ABB RAPID module: FSNA0464C.mod

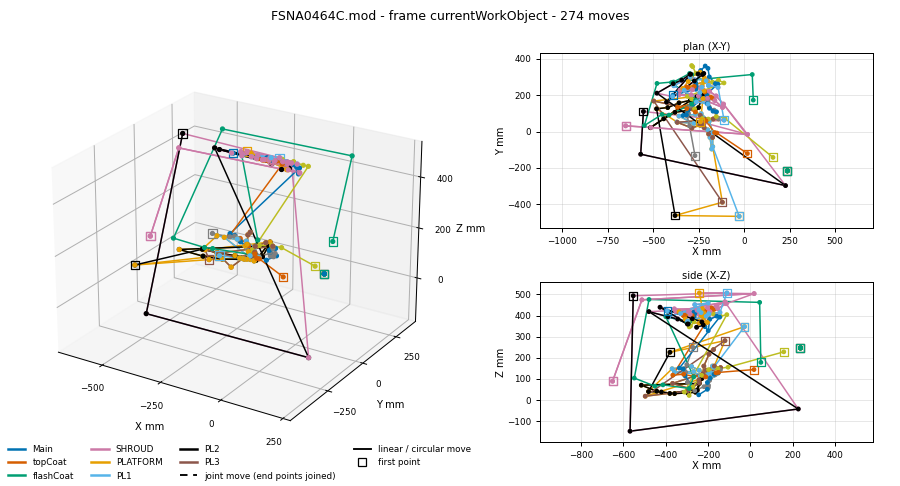
[picture p0: tool path of FSNA0464C.mod in frame currentWorkObject, 274 of 274 moves have a stored position in this frame; points joined in program order, loops and branches not executed]
MODULE FSNA0464C

    ! 10-10-24
    !
    ! declare and/or define variables that are local to this module
    LOCAL CONST listitem partProgram{3}:=[["","TopCoat"],["","FlashCoat"],[stEmpty,"Stop"]];
    LOCAL VAR string defaultValueString;
    VAR num itemselected:=0;
    VAR buttondata buttonAnswer:=0;
    LOCAL VAR robtarget pInt_temp1;
	PERS zonedata pathairfoil:=[FALSE,100,100,100,75,75,15];
    !
    VAR num myTemp := 0;
    VAR num X_Shift := 0;
    VAR num X_Value := 0;
    VAR num Y_Shift := 0;
    VAR num Y_Value := 0;
    VAR num Z_Shift := 0;
    VAR num Z_Value := 0;
    VAR num Speed := 0;
    VAR num LargestDistance := 0;
    VAR num numberOfLines := 0;
    VAR num FirstPass := 0;
    !
    ! positions for Airfoil CTARR
    CONST robtarget p1:=[[-480.99,124.94,40.31],[0.241886,0.571759,0.755176,0.210457],[0,1,1,0],[0,67.5741,9E+9,9E+9,9E+9,9E+9]];
    CONST robtarget p2:=[[-419.82,131.58,38.25],[0.241885,0.571758,0.755177,0.210457],[0,1,1,0],[0,59.8741,9E+9,9E+9,9E+9,9E+9]];
    CONST robtarget p3:=[[-357.80,157.50,30.89],[0.25135,0.552212,0.746055,0.274387],[0,1,1,0],[0,49.8741,9E+9,9E+9,9E+9,9E+9]];
    CONST robtarget p4:=[[-295.67,171.59,34.02],[0.258412,0.447595,0.729271,0.448381],[0,1,1,0],[0,44.2741,9E+9,9E+9,9E+9,9E+9]];
    CONST robtarget p5:=[[-258.93,192.30,37.24],[0.258413,0.447594,0.729271,0.448381],[0,1,1,0],[0,30.6741,9E+9,9E+9,9E+9,9E+9]];
    CONST robtarget p6:=[[-240.79,207.18,79.11],[0.336518,0.448757,0.687079,0.461839],[0,1,1,0],[0,18.4741,9E+9,9E+9,9E+9,9E+9]];
    CONST robtarget p7:=[[1532.27,28.26,128.24],[0.245924,0.528851,0.800385,-0.138642],[0,0,0,0],[0,558.621,9E+9,9E+9,9E+9,9E+9]];
    CONST robtarget p8:=[[-514.99,21.05,70.50],[0.286821,0.504649,0.813028,0.0452658],[0,1,1,0],[0,67.5741,9E+9,9E+9,9E+9,9E+9]];
    CONST robtarget p9:=[[-441.94,69.98,41.95],[0.327155,0.53741,0.777145,0.0143071],[0,1,1,0],[0,59.8741,9E+9,9E+9,9E+9,9E+9]];
    CONST robtarget p10:=[[-380.23,105.47,31.38],[0.392331,0.6189,0.675982,0.078028],[0,2,1,0],[0,49.8741,9E+9,9E+9,9E+9,9E+9]];
    !
    CONST robtarget p11:=[[-268.27,122.31,50.17],[0.448624,0.648801,0.591368,0.167566],[0,2,1,0],[0,44.2741,9E+9,9E+9,9E+9,9E+9]];
    CONST robtarget p12:=[[-250.17,131.85,47.00],[0.481979,0.715929,0.422761,0.276432],[0,2,1,0],[0,30.6741,9E+9,9E+9,9E+9,9E+9]];
    CONST robtarget p13:=[[-229.13,197.03,101.76],[0.452914,0.539488,0.537819,0.463219],[0,1,1,0],[0,24.4741,9E+9,9E+9,9E+9,9E+9]];
    CONST robtarget p14:=[[1816.81,23.63,146.28],[0.530012,0.0601364,0.839977,0.0995457],[-1,0,-1,0],[0,485.704,9E+9,9E+9,9E+9,9E+9]];
    CONST robtarget p15:=[[1496.69,-77.72,540],[0.712477,-0.0505666,0.699591,0.0197792],[-1,-1,-1,0],[120.002,9E+09,9E+09,9E+09,9E+09,9E+09]];
    CONST robtarget p16:=[[1503.37,67.93,540],[0.712477,-0.0505667,0.699591,0.0197793],[-1,-1,-1,0],[150.003,9E+09,9E+09,9E+09,9E+09,9E+09]];
    CONST robtarget p17:=[[1525.14,108.88,540],[0.712477,-0.0505668,0.699591,0.0197793],[-1,-1,-1,0],[195.004,9E+09,9E+09,9E+09,9E+09,9E+09]];
    CONST robtarget p18:=[[1539.77,199.84,540],[0.712477,-0.0505668,0.699591,0.0197793],[-1,-1,-1,0],[230.001,9E+09,9E+09,9E+09,9E+09,9E+09]];
    CONST robtarget p19:=[[-172.56,-82.90,154.81],[0.0598896,-0.960037,0.272975,-0.0150686],[0,-1,2,0],[0,162.3,9E+9,9E+9,9E+9,9E+9]];
    CONST robtarget p20:=[[-172.53,-7.13,117.30],[0.0598902,-0.960037,0.272975,-0.0150687],[0,-1,2,0],[0,164,9E+9,9E+9,9E+9,9E+9]];
    !
    CONST robtarget p21:=[[-191.10,57.42,100.93],[0.0655881,-0.94736,0.311192,-0.0369689],[0,-1,2,0],[0,173.5,9E+9,9E+9,9E+9,9E+9]];
    CONST robtarget p22:=[[-236.16,98.35,113.48],[0.0598898,-0.960037,0.272975,-0.0150686],[0,-1,2,0],[0,188.8,9E+9,9E+9,9E+9,9E+9]];
    CONST robtarget p23:=[[-267.77,93.84,135.02],[0.0372043,-0.989337,0.123334,0.0679511],[0,-1,2,0],[0,200.8,9E+9,9E+9,9E+9,9E+9]];
    CONST robtarget p24:=[[-358.18,84.85,132.45],[0.0372035,-0.989337,0.123334,0.0679511],[0,-1,2,0],[0,209.5,9E+9,9E+9,9E+9,9E+9]];
    CONST robtarget p25:=[[-172.53,-7.13,117.30],[0.0598902,-0.960037,0.272975,-0.0150687],[0,-1,2,0],[0,164,9E+9,9E+9,9E+9,9E+9]];
    CONST robtarget p26:=[[-178.25,-95.93,161.15],[0.0598899,-0.960037,0.272975,-0.0150685],[0,-1,2,0],[0,162.3,9E+9,9E+9,9E+9,9E+9]];
    CONST robtarget p27:=[[-187.56,-32.42,129.52],[0.0598899,-0.960037,0.272975,-0.0150687],[0,-1,2,0],[0,164,9E+9,9E+9,9E+9,9E+9]];
    CONST robtarget p28:=[[-200.37,9.66,124.39],[0.065588,-0.94736,0.311192,-0.0369689],[0,-1,2,0],[0,173.5,9E+9,9E+9,9E+9,9E+9]];
    CONST robtarget p29:=[[-241.64,42.37,141.08],[0.05989,-0.960037,0.272975,-0.0150686],[0,-1,2,0],[0,188.8,9E+9,9E+9,9E+9,9E+9]];
    CONST robtarget p30:=[[-277.12,44.60,159.21],[0.037204,-0.989337,0.123334,0.0679512],[0,-1,2,0],[0,200.8,9E+9,9E+9,9E+9,9E+9]];
    !
    CONST robtarget p31:=[[-369.35,52.61,148.19],[0.0372036,-0.989337,0.123334,0.0679511],[0,-1,2,0],[0,209.5,9E+9,9E+9,9E+9,9E+9]];
    CONST robtarget p32:=[[1621.31,158.58,690],[0.712477,-0.0505667,0.699591,0.0197792],[-1,-1,-1,0],[-0.00322896,9E+09,9E+09,9E+09,9E+09,9E+09]];
    CONST robtarget p33:=[[1620.84,58.68,700],[0.712477,-0.0505667,0.699591,0.0197793],[-1,-1,-1,0],[9.9958,9E+09,9E+09,9E+09,9E+09,9E+09]];
    CONST robtarget p34:=[[1665.7,-160.7,700],[0.712477,-0.0505667,0.699591,0.0197793],[-1,-1,-1,0],[70.0029,9E+09,9E+09,9E+09,9E+09,9E+09]];
    CONST robtarget p35:=[[1496.69,-77.72,700],[0.712477,-0.0505666,0.699591,0.0197792],[-1,-1,-1,0],[120.002,9E+09,9E+09,9E+09,9E+09,9E+09]];
    CONST robtarget p36:=[[1503.37,67.93,690],[0.712477,-0.0505667,0.699591,0.0197793],[-1,-1,-1,0],[150.003,9E+09,9E+09,9E+09,9E+09,9E+09]];
    CONST robtarget p37:=[[1525.14,108.88,690],[0.712477,-0.0505668,0.699591,0.0197793],[-1,-1,-1,0],[195.004,9E+09,9E+09,9E+09,9E+09,9E+09]];
    CONST robtarget p38:=[[1539.77,199.84,700],[0.712477,-0.0505668,0.699591,0.0197793],[-1,-1,-1,0],[230.001,9E+09,9E+09,9E+09,9E+09,9E+09]];
    CONST robtarget p39:=[[1444.86,284.59,700],[0.712477,-0.0505668,0.699591,0.0197793],[0,-1,-1,0],[270.004,9E+09,9E+09,9E+09,9E+09,9E+09]];
    CONST robtarget p40:=[[-496.31,167.54,18.41],[0.302398,0.557141,0.772704,0.0328229],[0,1,1,0],[0,35.3741,9E+9,9E+9,9E+9,9E+9]];
    !
    CONST robtarget p41:=[[-296.07,126.18,42.89],[0.3024,0.55714,0.772704,0.0328239],[0,1,1,0],[0,25.4741,9E+9,9E+9,9E+9,9E+9]];
    CONST robtarget p42:=[[-240.83,89.12,81.91],[0.302399,0.557141,0.772704,0.0328236],[-1,1,1,0],[0,4.4741,9E+9,9E+9,9E+9,9E+9]];
    CONST robtarget p43:=[[-215.91,67.47,112.59],[0.302399,0.557141,0.772704,0.0328236],[-1,1,1,0],[0,-9.7259,9E+9,9E+9,9E+9,9E+9]];
    CONST robtarget p44:=[[-208.79,59.37,141.39],[0.302399,0.557141,0.772704,0.0328237],[-1,1,1,0],[0,-25.4259,9E+9,9E+9,9E+9,9E+9]];
    CONST robtarget p45:=[[-169.72,69.14,160.90],[0.302399,0.557141,0.772704,0.0328238],[-1,1,1,0],[0,-33.5259,9E+9,9E+9,9E+9,9E+9]];
    CONST robtarget p46:=[[-140.26,69.36,153.83],[0.302399,0.55714,0.772704,0.0328239],[-1,1,1,0],[0,-42.5259,9E+9,9E+9,9E+9,9E+9]];
    CONST robtarget p48:=[[-366.97,50.44,78.97],[0.302398,0.557141,0.772704,0.0328232],[0,1,1,0],[0,35.3741,9E+9,9E+9,9E+9,9E+9]];
    CONST robtarget p49:=[[-287.06,19.27,54.47],[0.302399,0.557141,0.772704,0.032823],[-1,1,1,0],[0,25.4741,9E+9,9E+9,9E+9,9E+9]];

    PERS robtarget p201:=[[-190.59,221.15,418.28],[0.323876,-0.134268,0.48472,0.801326],[-1,1,0,0],[0,-184.719,9E+9,9E+9,9E+9,9E+9]];
    PERS robtarget p202:=[[-238.99,240.86,403.58],[0.323876,-0.134268,0.48472,0.801326],[-1,1,0,0],[0,-184.719,9E+9,9E+9,9E+9,9E+9]];
    PERS robtarget p203:=[[-283.49,230.19,405.56],[0.323876,-0.134268,0.48472,0.801326],[-1,1,0,0],[0,-184.719,9E+9,9E+9,9E+9,9E+9]];
    PERS robtarget p204:=[[-351.84,227.15,419.55],[0.323876,-0.134268,0.48472,0.801326],[-1,1,0,0],[0,-184.719,9E+9,9E+9,9E+9,9E+9]];
    PERS robtarget p205:=[[-138.38,318.26,282.97],[0.820959,-0.00154933,0.553533,0.14009],[0,2,-2,0],[0,-333.4,9E+9,9E+9,9E+9,9E+9]];
    PERS robtarget p206:=[[1522.85,30.49,127.90],[0.693528,-0.018539,0.719901,0.0204515],[-1,-1,-1,0],[0,525.079,9E+9,9E+9,9E+9,9E+9]];
    PERS robtarget p207:=[[1533.71,58.37,146.07],[0.688077,-0.0919601,0.714028,0.0908723],[-1,-1,-1,0],[0,525.079,9E+9,9E+9,9E+9,9E+9]];
    PERS robtarget p208:=[[-118.63,132.39,464.09],[0.341814,-0.118033,0.331132,0.871541],[-1,1,0,0],[0,-184.719,9E+9,9E+9,9E+9,9E+9]];
    PERS robtarget p209:=[[-161.24,170.27,444.44],[0.34262,-0.116882,0.321021,0.875155],[-1,1,0,0],[0,-184.719,9E+9,9E+9,9E+9,9E+9]];
    PERS robtarget p210:=[[-201.32,182.62,436.33],[0.342259,-0.117406,0.32561,0.873529],[-1,1,0,0],[0,-184.719,9E+9,9E+9,9E+9,9E+9]];
    !
    PERS robtarget p211:=[[-251.52,195.90,424.71],[0.34323,-0.11596,0.312977,0.877948],[-1,1,0,0],[0,-184.719,9E+9,9E+9,9E+9,9E+9]];
    PERS robtarget p212:=[[-291.38,201.77,418.66],[0.342305,-0.117339,0.325025,0.873738],[-1,1,0,0],[0,-184.719,9E+9,9E+9,9E+9,9E+9]];
    PERS robtarget p213:=[[-358.88,201.75,431.17],[0.34234,-0.11729,0.324591,0.873892],[-1,1,0,0],[0,-184.719,9E+9,9E+9,9E+9,9E+9]];
    PERS robtarget p214:=[[1526.81,49.01,147.72],[0.53358,0.309144,0.772491,-0.151589],[0,0,0,0],[0,525.079,9E+9,9E+9,9E+9,9E+9]];
    PERS robtarget p215:=[[-141.45,-101.58,920.03],[0.650986,0.194184,0.706774,-0.197436],[-1,0,0,0],[82.817,9E+09,9E+09,9E+09,9E+09,9E+09]];
    PERS robtarget p216:=[[-88.05,-18.09,920.70],[0.650993,0.194178,0.706763,-0.197458],[0,0,0,0],[82.817,9E+09,9E+09,9E+09,9E+09,9E+09]];
    PERS robtarget p217:=[[-21.87,98.95,918.25],[0.65099,0.194168,0.706777,-0.197427],[0,0,0,0],[82.817,9E+09,9E+09,9E+09,9E+09,9E+09]];
    PERS robtarget p218:=[[53.24,222.48,897.26],[0.65098,0.194179,0.706786,-0.197419],[0,0,0,0],[82.817,9E+09,9E+09,9E+09,9E+09,9E+09]];
    PERS robtarget p219:=[[45.58,94.46,899.85],[0.0855565,0.697288,0.707868,-0.0734352],[0,0,0,0],[104.005,9E+09,9E+09,9E+09,9E+09,9E+09]];
    PERS robtarget p220:=[[-221.03,177.90,433.71],[0.343488,0.0801029,0.438498,0.826631],[-1,1,0,0],[0,-140.019,9E+9,9E+9,9E+9,9E+9]];
    !
    PERS robtarget p221:=[[-226.19,180.94,432.49],[0.55509,0.111637,0.37794,0.732512],[0,1,0,0],[0,-140.019,9E+9,9E+9,9E+9,9E+9]];
    PERS robtarget p222:=[[-219.63,223.62,412.03],[0.561411,0.0905932,0.427662,0.702649],[0,1,0,0],[0,-140.019,9E+9,9E+9,9E+9,9E+9]];
    PERS robtarget p223:=[[-230.74,249.72,398.97],[0.562161,0.0874597,0.434857,0.698015],[0,1,0,0],[0,-140.019,9E+9,9E+9,9E+9,9E+9]];
    PERS robtarget p224:=[[-220.10,274.50,389.30],[0.52604,0.192483,0.577288,0.594113],[0,1,0,0],[0,-140.019,9E+9,9E+9,9E+9,9E+9]];
    PERS robtarget p225:=[[-202.24,278.15,367.26],[0.464891,0.348117,0.609092,0.540091],[0,1,1,0],[0,-140.019,9E+9,9E+9,9E+9,9E+9]];
    PERS robtarget p226:=[[1608.55,16.90,696.10],[0.496587,-0.139785,0.281765,-0.808993],[0,-1,1,0],[25.0035,9E+9,9E+9,9E+9,9E+9,9E+9]];
    PERS robtarget p227:=[[1502.42,-81.35,694.68],[0.496587,-0.139785,0.281765,-0.808993],[0,-1,1,0],[0,9E+9,9E+9,9E+9,9E+9,9E+9]];
    PERS robtarget p228:=[[1461.90,-160.07,687.75],[0.496587,-0.139785,0.281765,-0.808993],[0,-1,1,0],[-0.000826709,9E+9,9E+9,9E+9,9E+9,9E+9]];
    !
    PERS robtarget p231:=[[-293.61,298.88,371.24],[0.0151509,-0.0827354,0.608731,0.788906],[-1,0,0,0],[0,-140.019,9E+9,9E+9,9E+9,9E+9]];
    PERS robtarget p232:=[[-241.43,325.70,363.53],[0.174125,0.0732031,0.694697,0.694059],[-1,0,0,0],[0,-140.019,9E+9,9E+9,9E+9,9E+9]];
    PERS robtarget p233:=[[-219.10,295.28,358.44],[0.464891,0.348117,0.609092,0.540091],[0,1,1,0],[0,-140.019,9E+9,9E+9,9E+9,9E+9]];
    PERS robtarget p234:=[[1381.21,176.71,690.45],[0.509919,-0.0782388,0.181097,-0.837296],[0,-1,1,0],[74.9967,9E+9,9E+9,9E+9,9E+9,9E+9]];
    PERS robtarget p235:=[[1460.37,118.23,690.06],[0.505886,-0.101083,0.218555,-0.828308],[0,-1,1,0],[49.9958,9E+9,9E+9,9E+9,9E+9,9E+9]];
    PERS robtarget p236:=[[1453.88,16.90,696.10],[0.496587,-0.139785,0.281765,-0.808993],[0,-1,1,0],[25.0035,9E+9,9E+9,9E+9,9E+9,9E+9]];
    PERS robtarget p237:=[[1308.94,-160.07,687.75],[0.496587,-0.139785,0.281765,-0.808993],[0,-1,1,0],[-0.000826709,9E+9,9E+9,9E+9,9E+9,9E+9]];
    PERS robtarget p238:=[[1411.45,-160.07,687.75],[0.496587,-0.139785,0.281765,-0.808993],[0,-1,1,0],[-0.000826709,9E+9,9E+9,9E+9,9E+9,9E+9]];
    !
    PERS robtarget p241:=[[1858.30,301.74,499.76],[0.179089,0.917392,0.34153,0.0983641],[0,1,0,0],[-175.061,9E+9,9E+9,9E+9,9E+9,9E+9]];
    PERS robtarget p242:=[[1614.86,199.00,509.29],[0.175594,0.951771,0.23609,0.086952],[0,1,-1,0],[-190.061,9E+9,9E+9,9E+9,9E+9,9E+9]];
    PERS robtarget p243:=[[1502.55,134.04,503.05],[0.185136,0.908581,0.362955,0.0920279],[0,1,0,0],[-220.061,9E+9,9E+9,9E+9,9E+9,9E+9]];
    PERS robtarget p244:=[[1494.58,104.81,490.86],[0.174159,0.800358,0.560783,0.120907],[0,1,0,0],[-240.061,9E+9,9E+9,9E+9,9E+9,9E+9]];
    PERS robtarget p245:=[[1559.49,159.93,488.36],[0.149738,0.674434,0.699604,0.182406],[0,1,0,0],[-310.061,9E+9,9E+9,9E+9,9E+9,9E+9]];
    PERS robtarget p246:=[[1600.54,33.00,493.44],[0.172748,0.593565,0.769913,0.158344],[-1,0,0,0],[-330.061,9E+9,9E+9,9E+9,9E+9,9E+9]];
    PERS robtarget p247:=[[1500.24,-78.88,512.52],[0.130233,0.625317,0.75886,0.12708],[-1,0,0,0],[-350.061,9E+9,9E+9,9E+9,9E+9,9E+9]];
    PERS robtarget p248:=[[1338.41,-93.31,512.24],[0.126705,0.803062,0.571687,0.110503],[-1,1,0,0],[-375.061,9E+9,9E+9,9E+9,9E+9,9E+9]];
    !

    ! declare and/or define position variables that are local to this module
	PERS robtarget home:=[[114.84,-94.02,-57.43],[0.398229,-0.576485,0.66735,0.252432],[-1,-1,-1,0],[0,372.2,9E+9,9E+9,9E+9,9E+9]];
	PERS robtarget pounce:=[[114.84,-94.02,-57.43],[0.398229,-0.576485,0.66735,0.252432],[-1,-1,-1,0],[0,0,9E+9,9E+9,9E+9,9E+9]];
    PERS robtarget home10:=[[-37.25,141.01,1171.15],[0.656992,0.226174,0.64921,-0.309408],[0,-1,0,0],[-0.00177226,9E+09,9E+09,9E+09,9E+09,9E+09]];
    PERS robtarget home20:=[[-47.87,162.56,920.76],[0.566373,0.264704,0.729584,-0.277237],[0,0,0,0],[0.0306373,9E+09,9E+09,9E+09,9E+09,9E+09]];
    PERS robtarget pounce10:=[[1506.92,-117.30,148.10],[0.362896,-0.228602,0.902396,0.0415831],[-1,-1,-1,0],[0,-6.2069,9E+9,9E+9,9E+9,9E+9]];
    PERS robtarget mypounce:=[[-379.47,-461.24,226.09],[0.186927,-0.20553,0.960411,0.0206579],[-1,0,1,0],[0,162.3,9E+9,9E+9,9E+9,9E+9]];
    PERS robtarget mypounce10:=[[-27.24,-465.79,347.27],[0.059889,-0.960037,0.272975,-0.0150683],[-1,-1,2,0],[0,162.3,9E+9,9E+9,9E+9,9E+9]];
    PERS robtarget mypounce20:=[[-119.56,-388.27,281.05],[0.286821,0.504649,0.813028,0.0452658],[-1,1,1,0],[0,67.5741,9E+9,9E+9,9E+9,9E+9]];
    PERS robtarget mypounce30:=[[158.59,-142.09,228.20],[0.41173,-0.607554,0.614434,0.289531],[-1,-1,1,0],[0,-21.0832,9E+9,9E+9,9E+9,9E+9]];
    PERS robtarget mypounce40:=[[-391.18,199.72,419.59],[0.346718,-0.644484,0.557145,0.39245],[0,-1,1,0],[0,-99.7753,9E+9,9E+9,9E+9,9E+9]];
    PERS robtarget mypounce50:=[[17.77,-120.71,144.39],[0.403174,-0.614096,0.639379,0.227004],[-1,-1,2,0],[0,-195,9E+9,9E+9,9E+9,9E+9]];
    PERS wobjdata wobj1:=[FALSE,TRUE,"",[[0,0,0],[1,0,0,0]],[[1526.4,-255.043,47.4813],[0.766931,0.185105,-0.133095,-0.599865]]];
    PERS robtarget p0:=[[1402.40,207.74,74.69],[0.420282,-0.489062,0.761608,-0.0643041],[0,-1,0,0],[0,453.104,9E+9,9E+9,9E+9,9E+9]];
    PERS robtarget mypounce60:=[[50.15,172.68,178.39],[0.441257,-0.541665,0.672728,0.243575],[-1,0,1,0],[0,-286.004,9E+9,9E+9,9E+9,9E+9]];
    PERS robtarget tempval:=[[1776.74,50.33,181.37],[0.419919,-0.484892,0.74874,-0.167142],[-1,-1,0,0],[0,453.104,9E+9,9E+9,9E+9,9E+9]];
    PERS robtarget tempval10:=[[1776.74,50.33,181.37],[0.419919,-0.484892,0.74874,-0.167142],[-1,-1,0,0],[0,453.104,9E+9,9E+9,9E+9,9E+9]];
    PERS robtarget mypouncePL:=[[1450.05,-296.49,158.45],[0.000887637,0.674822,0.737972,0.00347664],[-1,0,0,0],[0,368.4,9E+9,9E+9,9E+9,9E+9]];
    PERS robtarget mypouncePL10:=[[1453.74,-212.15,169.09],[0.000887898,0.674822,0.737972,0.00347632],[-1,0,0,0],[0,368.4,9E+9,9E+9,9E+9,9E+9]];
    PERS robtarget p50:=[[-242.82,35.16,96.19],[0.302399,0.557141,0.772704,0.0328234],[-1,1,1,0],[0,4.4741,9E+9,9E+9,9E+9,9E+9]];
    PERS robtarget p60:=[[-104.77,71.85,155.57],[0.235728,-0.65255,0.702889,0.15671],[-1,-1,1,0],[0,-21.0832,9E+9,9E+9,9E+9,9E+9]];
    PERS robtarget p70:=[[-223.35,269.54,407.36],[0.490279,-0.512469,0.629658,0.317069],[0,0,2,0],[0,-21.0832,9E+9,9E+9,9E+9,9E+9]];
    PERS robtarget p51:=[[-224.08,37.20,124.71],[0.302399,0.557141,0.772704,0.0328239],[-1,1,1,0],[0,-9.7259,9E+9,9E+9,9E+9,9E+9]];
    PERS robtarget p53:=[[-195.00,-13.72,216.84],[0.302399,0.55714,0.772704,0.0328239],[-1,1,1,0],[0,-33.5259,9E+9,9E+9,9E+9,9E+9]];
    PERS robtarget p52:=[[-219.36,20.60,161.04],[0.302399,0.557141,0.772704,0.0328233],[-1,1,1,0],[0,-25.4259,9E+9,9E+9,9E+9,9E+9]];
    PERS robtarget p54:=[[-173.44,-32.53,238.99],[0.302399,0.55714,0.772704,0.0328235],[-1,1,1,0],[0,-42.5259,9E+9,9E+9,9E+9,9E+9]];
    PERS robtarget p55:=[[1627.55,-144.85,103.80],[0.37608,-0.272238,0.874139,0.142592],[-1,-1,-1,0],[0,473.679,9E+9,9E+9,9E+9,9E+9]];
    PERS robtarget p56:=[[1636.24,-58.87,104.20],[0.37057,-0.304807,0.863301,0.156466],[-1,-1,-1,0],[0,473.679,9E+9,9E+9,9E+9,9E+9]];
    PERS robtarget p57:=[[1542.81,-38.49,90.01],[0.365729,-0.330862,0.853641,0.167539],[-1,-1,-1,0],[0,473.679,9E+9,9E+9,9E+9,9E+9]];
    PERS robtarget p58:=[[1415.80,3.28,64.46],[0.365729,-0.330862,0.853641,0.167539],[-1,-1,-1,0],[0,473.679,9E+9,9E+9,9E+9,9E+9]];
    PERS robtarget p67:=[[-110.76,267.07,404.11],[0.363074,-0.624312,0.643864,0.252685],[-1,-1,1,0],[0,-21.0832,9E+9,9E+9,9E+9,9E+9]];
    PERS robtarget p61:=[[-152.80,82.65,148.87],[0.187257,-0.658057,0.719316,0.120335],[0,-1,1,0],[0,-21.0832,9E+9,9E+9,9E+9,9E+9]];
    PERS robtarget p62:=[[-197.09,68.49,143.85],[0.187257,-0.658057,0.719316,0.120335],[0,-1,1,0],[0,-21.0832,9E+9,9E+9,9E+9,9E+9]];
    PERS robtarget p63:=[[-229.45,71.30,117.03],[0.227436,-0.599619,0.763307,0.0780525],[0,0,2,0],[0,-21.0832,9E+9,9E+9,9E+9,9E+9]];
    PERS robtarget p80:=[[-265.55,232.07,416.89],[0.144535,-0.701198,0.368316,0.593105],[-1,0,1,0],[0,-99.7753,9E+9,9E+9,9E+9,9E+9]];
    PERS robtarget p81:=[[-261.58,246.21,409.97],[0.144535,-0.701198,0.368316,0.593105],[-1,0,1,0],[0,-99.7753,9E+9,9E+9,9E+9,9E+9]];
    PERS robtarget p82:=[[-265.06,264.67,396.52],[0.144535,-0.701198,0.368316,0.593105],[-1,0,1,0],[0,-99.7753,9E+9,9E+9,9E+9,9E+9]];
    PERS robtarget p83:=[[-238.77,335.25,363.62],[0.339406,-0.656714,0.470947,0.481392],[-1,-1,1,0],[0,-99.7753,9E+9,9E+9,9E+9,9E+9]];
    PERS robtarget p93:=[[-202.77,199.89,50.99],[0.336532,-0.904926,0.260301,-0.00990511],[0,-1,2,0],[0,-99.7753,9E+9,9E+9,9E+9,9E+9]];
    PERS robtarget p103:=[[-267.84,107.34,111.99],[0.393028,-0.576819,0.672319,0.246569],[0,0,2,0],[0,-195,9E+9,9E+9,9E+9,9E+9]];
    PERS robtarget p94:=[[-202.59,152.76,83.34],[0.304048,-0.849853,0.395123,-0.170828],[0,-1,2,0],[0,-99.7753,9E+9,9E+9,9E+9,9E+9]];
    PERS robtarget p84:=[[-213.83,359.92,347.10],[0.394944,-0.635518,0.506567,0.4284],[-1,-1,1,0],[0,-99.7753,9E+9,9E+9,9E+9,9E+9]];
    PERS robtarget p85:=[[-198.67,346.90,328.05],[0.475693,-0.58931,0.583419,0.293345],[0,-1,2,0],[0,-99.7753,9E+9,9E+9,9E+9,9E+9]];
    PERS robtarget p95:=[[-190.25,127.73,103.49],[0.304048,-0.849853,0.395123,-0.170828],[0,-1,2,0],[0,-99.7753,9E+9,9E+9,9E+9,9E+9]];
    PERS robtarget p105:=[[-366.09,132.79,118.09],[0.323041,-0.635333,0.624263,0.319831],[0,-1,1,0],[0,-195,9E+9,9E+9,9E+9,9E+9]];
    PERS robtarget p86:=[[-191.26,300.09,382.38],[0.59614,-0.483857,0.607528,0.203491],[0,-1,2,0],[0,-99.7753,9E+9,9E+9,9E+9,9E+9]];
    PERS robtarget p87:=[[-157.75,263.05,396.69],[0.59614,-0.483857,0.607528,0.203491],[0,-1,2,0],[0,-99.7753,9E+9,9E+9,9E+9,9E+9]];
    PERS robtarget p97:=[[-151.71,108.34,127.85],[0.455068,-0.790762,0.388826,-0.128156],[0,-1,2,0],[0,-99.7753,9E+9,9E+9,9E+9,9E+9]];
    PERS robtarget p107:=[[-171.00,182.73,428.83],[0.510833,-0.489852,0.656726,0.260396],[0,0,2,0],[0,-195,9E+9,9E+9,9E+9,9E+9]];
    PERS robtarget p88:=[[-144.63,260.94,392.22],[0.53853,-0.525652,0.641502,0.148831],[0,-1,2,0],[0,-99.7753,9E+9,9E+9,9E+9,9E+9]];
    PERS robtarget p89:=[[-335.05,88.30,151.37],[0.225425,-0.851908,0.331482,0.336981],[0,-1,2,0],[0,-99.7753,9E+9,9E+9,9E+9,9E+9]];
    PERS robtarget p68:=[[-140.93,282.02,396.74],[0.416985,-0.58835,0.652857,0.231831],[0,-1,2,0],[0,-21.0832,9E+9,9E+9,9E+9,9E+9]];
    PERS robtarget p59:=[[1256.15,38.08,77.18],[0.365729,-0.330862,0.853641,0.167539],[-1,-1,-1,0],[0,473.679,9E+9,9E+9,9E+9,9E+9]];
    PERS robtarget p47:=[[1532.27,28.26,128.24],[0.245924,0.528851,0.800385,-0.138642],[0,0,0,0],[0,558.621,9E+9,9E+9,9E+9,9E+9]];
    PERS robtarget p90:=[[-316.97,91.92,146.99],[0.220546,-0.85345,0.324574,0.342979],[-1,-1,2,0],[0,-99.7753,9E+9,9E+9,9E+9,9E+9]];
    PERS robtarget p66:=[[-311.42,193.18,37.97],[0.305868,-0.633875,0.658667,0.266093],[0,-1,1,0],[0,-21.0832,9E+9,9E+9,9E+9,9E+9]];
    PERS robtarget p64:=[[-272.18,123.81,60.95],[0.271775,-0.59184,0.749775,0.117051],[0,0,2,0],[0,-21.0832,9E+9,9E+9,9E+9,9E+9]];
    PERS robtarget p65:=[[-288.87,179.42,22.10],[0.318069,-0.603467,0.699672,0.212409],[0,0,2,0],[0,-21.0832,9E+9,9E+9,9E+9,9E+9]];
    PERS robtarget p69:=[[-175.57,271.09,407.55],[0.490279,-0.512469,0.629658,0.317069],[0,0,2,0],[0,-21.0832,9E+9,9E+9,9E+9,9E+9]];
    PERS robtarget p71:=[[-265.49,320.04,370.00],[0.469908,-0.52339,0.645441,0.29775],[0,0,2,0],[0,-21.0832,9E+9,9E+9,9E+9,9E+9]];
    PERS robtarget p72:=[[-282.33,355.82,350.44],[0.500121,-0.506862,0.621602,0.326466],[0,0,2,0],[0,-21.0832,9E+9,9E+9,9E+9,9E+9]];
    PERS robtarget p73:=[[-288.32,362.58,346.09],[0.324166,-0.650206,0.573552,0.3784],[0,-1,1,0],[0,-21.0832,9E+9,9E+9,9E+9,9E+9]];
    PERS robtarget home30:=[[237.33,-215.55,246.81],[0.488992,-0.630948,0.551207,0.242821],[-1,-1,2,0],[0,0.0198783,9E+9,9E+9,9E+9,9E+9]];
    PERS robtarget mypounce70:=[[-512.28,22.13,474.14],[0.177753,-0.1662,0.259277,0.934643],[-1,1,0,0],[0,-286.004,9E+9,9E+9,9E+9,9E+9]];
    PERS robtarget p92:=[[-243.60,195.18,25.06],[0.170318,-0.924324,0.32307,0.110644],[0,-1,2,0],[0,-99.7753,9E+9,9E+9,9E+9,9E+9]];
    PERS robtarget p102:=[[-210.14,59.62,109.88],[0.401472,-0.568723,0.677656,0.236976],[0,0,2,0],[0,-195,9E+9,9E+9,9E+9,9E+9]];
    PERS robtarget p91:=[[-308.15,116.66,114.63],[0.186778,-0.861437,0.276725,0.382705],[-1,-1,2,0],[0,-99.7753,9E+9,9E+9,9E+9,9E+9]];
    PERS robtarget p100:=[[-150.03,-8.14,130.97],[0.440559,-0.527824,0.70084,0.190087],[0,0,2,0],[0,-195,9E+9,9E+9,9E+9,9E+9]];
    PERS robtarget p101:=[[-162.38,-5.44,129.39],[0.440559,-0.527824,0.70084,0.190087],[0,0,2,0],[0,-195,9E+9,9E+9,9E+9,9E+9]];
    PERS robtarget p104:=[[-314.86,126.21,122.37],[0.323041,-0.635333,0.624263,0.319831],[0,-1,1,0],[0,-195,9E+9,9E+9,9E+9,9E+9]];
    PERS robtarget p106:=[[-129.79,110.40,70.28],[0.403174,-0.614096,0.639379,0.227004],[-1,-1,0,0],[0,-66.5,9E+9,9E+9,9E+9,9E+9]];
    PERS robtarget p108:=[[-183.32,189.82,436.24],[0.510833,-0.489852,0.656726,0.260396],[0,0,2,0],[0,-195,9E+9,9E+9,9E+9,9E+9]];
    PERS robtarget p109:=[[-215.24,218.27,420.10],[0.461021,-0.542852,0.639298,0.289947],[0,0,2,0],[0,-195,9E+9,9E+9,9E+9,9E+9]];
    PERS robtarget p110:=[[-274.07,247.53,399.54],[0.4533,-0.55171,0.633072,0.298923],[0,-1,2,0],[0,-195,9E+9,9E+9,9E+9,9E+9]];
    PERS robtarget p111:=[[-308.35,242.58,400.78],[0.403101,-0.611548,0.566935,0.376966],[0,-1,1,0],[0,-195,9E+9,9E+9,9E+9,9E+9]];
    PERS robtarget p112:=[[-316.07,243.83,398.93],[0.372437,-0.628259,0.548013,0.407754],[0,-1,1,0],[0,-195,9E+9,9E+9,9E+9,9E+9]];
    PERS robtarget p113:=[[-22.45,-122.19,118.26],[0.403174,-0.614096,0.639379,0.227004],[-1,-1,0,0],[0,-195,9E+9,9E+9,9E+9,9E+9]];
    PERS robtarget p123:=[[-266.87,171.99,110.22],[0.39541,-0.58203,0.646346,0.295174],[0,0,2,0],[0,-286.004,9E+9,9E+9,9E+9,9E+9]];
    PERS robtarget p120:=[[-451.03,94.08,66.05],[0.230357,-0.682791,0.531307,0.445472],[0,-1,1,0],[0,-286.004,9E+9,9E+9,9E+9,9E+9]];
    PERS robtarget p121:=[[-412.72,90.37,72.14],[0.202711,-0.694159,0.509558,0.466264],[0,-1,1,0],[0,-286.004,9E+9,9E+9,9E+9,9E+9]];
    PERS robtarget p131:=[[-407.31,65.48,14.57],[0.422742,-0.506784,0.679012,0.321562],[-1,1,-2,0],[0,-282,9E+9,9E+9,9E+9,9E+9]];
    PERS robtarget p122:=[[-288.57,151.17,55.23],[0.31947,-0.636015,0.596851,0.370394],[0,-1,1,0],[0,-286.004,9E+9,9E+9,9E+9,9E+9]];
    PERS robtarget mypounce80:=[[-292.56,139.70,-25.36],[0.403174,-0.614096,0.639379,0.227004],[-1,-1,0,0],[0,-24,9E+9,9E+9,9E+9,9E+9]];
    PERS robtarget tp10:=[[-292.56,139.70,-25.36],[0.403174,-0.614096,0.639379,0.227004],[-1,-1,0,0],[0,-24,9E+9,9E+9,9E+9,9E+9]];
    !
    PERS robtarget mypounce110:=[[-482.41,64.04,89.43],[0.313843,-0.686244,0.567806,0.32889],[-1,-1,-1,0],[0,-31.4,9E+9,9E+9,9E+9,9E+9]];
    PERS robtarget p560:=[[-186.00,20.77,115.70],[0.313843,-0.686244,0.567806,0.32889],[-1,-1,-1,0],[0,-31.4,9E+9,9E+9,9E+9,9E+9]];
    PERS robtarget p561:=[[-186.00,20.77,115.70],[0.313843,-0.686244,0.567806,0.32889],[-1,-1,-1,0],[0,-24.7,9E+9,9E+9,9E+9,9E+9]];
    PERS robtarget p562:=[[-184.82,16.87,78.50],[0.313843,-0.686244,0.567806,0.32889],[-1,-1,-1,0],[0,6,9E+9,9E+9,9E+9,9E+9]];
    PERS robtarget p563:=[[-180.94,54.11,26.07],[0.313843,-0.686244,0.567806,0.32889],[-1,-1,-1,0],[0,60,9E+9,9E+9,9E+9,9E+9]];
    PERS robtarget p564:=[[-216.60,41.81,21.25],[0.313843,-0.686244,0.567806,0.32889],[-1,-1,-1,0],[0,108,9E+9,9E+9,9E+9,9E+9]];
    PERS robtarget p565:=[[-127.38,57.13,98.81],[0.403174,-0.614096,0.639379,0.227004],[-1,-1,0,0],[0,-24.7,9E+9,9E+9,9E+9,9E+9]];
    PERS robtarget p566:=[[-189.86,194.53,362.31],[0.403174,-0.614096,0.639379,0.227004],[-1,-1,-1,0],[0,-24.7,9E+9,9E+9,9E+9,9E+9]];
    PERS robtarget p569:=[[-194.35,212.02,353.83],[0.313843,-0.686244,0.567806,0.32889],[-1,-1,-1,0],[0,6,9E+9,9E+9,9E+9,9E+9]];
    PERS robtarget p567:=[[-175.65,149.52,386.03],[0.313843,-0.686244,0.567806,0.32889],[-1,-1,-1,0],[0,-31.4,9E+9,9E+9,9E+9,9E+9]];
    PERS robtarget p568:=[[-205.18,198.55,359.09],[0.313843,-0.686244,0.567806,0.32889],[-1,-1,-1,0],[0,-24.7,9E+9,9E+9,9E+9,9E+9]];
    PERS robtarget p570:=[[-192.85,243.24,335.35],[0.313843,-0.686244,0.567806,0.32889],[-1,-1,-1,0],[0,60,9E+9,9E+9,9E+9,9E+9]];
    PERS robtarget p571:=[[-228.38,214.17,338.21],[0.344401,-0.678774,0.547989,0.346931],[-1,-1,-1,0],[0,108,9E+9,9E+9,9E+9,9E+9]];
    PERS robtarget mypounce120:=[[-477.64,-74.92,-193.25],[0.313843,-0.686244,0.567806,0.32889],[-1,-1,0,0],[0,-31.4,9E+9,9E+9,9E+9,9E+9]];
    PERS robtarget mypounce130:=[[-59.04,-166.15,-141.34],[0.313843,-0.686244,0.567806,0.32889],[-1,-1,0,0],[0,-31.4,9E+9,9E+9,9E+9,9E+9]];
    PERS robtarget mypounce140:=[[-63.83,-26.70,142.30],[0.313843,-0.686244,0.567806,0.32889],[-1,-1,-1,0],[0,-31.4,9E+9,9E+9,9E+9,9E+9]];
    PERS robtarget mypounce90:=[[-284.25,-46.11,66.24],[0.0193857,-0.784247,0.616476,0.0673647],[-1,-1,-1,0],[0,102,9E+9,9E+9,9E+9,9E+9]];
    PERS robtarget p580:=[[-284.25,-46.11,66.24],[0.0193857,-0.784247,0.616476,0.0673647],[-1,-1,-1,0],[0,102,9E+9,9E+9,9E+9,9E+9]];
    PERS robtarget p589:=[[-284.25,-46.11,66.24],[0.0193857,-0.784247,0.616476,0.0673647],[-1,-1,-1,0],[0,102,9E+9,9E+9,9E+9,9E+9]];
    PERS robtarget p581:=[[-284.25,-46.11,66.24],[0.0193857,-0.784247,0.616476,0.0673647],[-1,-1,-1,0],[0,102,9E+9,9E+9,9E+9,9E+9]];
    PERS robtarget p582:=[[-284.25,-46.11,66.24],[0.0193857,-0.784247,0.616476,0.0673647],[-1,-1,-1,0],[0,102,9E+9,9E+9,9E+9,9E+9]];
    PERS robtarget p583:=[[-284.25,-46.11,66.24],[0.0193857,-0.784247,0.616476,0.0673647],[-1,-1,-1,0],[0,102,9E+9,9E+9,9E+9,9E+9]];
    PERS robtarget p584:=[[-284.25,-46.11,66.24],[0.0193857,-0.784247,0.616476,0.0673647],[-1,-1,-1,0],[0,102,9E+9,9E+9,9E+9,9E+9]];
    PERS robtarget p585:=[[-284.25,-46.11,66.24],[0.0193857,-0.784247,0.616476,0.0673647],[-1,-1,-1,0],[0,102,9E+9,9E+9,9E+9,9E+9]];
    PERS robtarget p586:=[[-284.25,-46.11,66.24],[0.0193857,-0.784247,0.616476,0.0673647],[-1,-1,-1,0],[0,102,9E+9,9E+9,9E+9,9E+9]];
    PERS robtarget p587:=[[-284.25,-46.11,66.24],[0.0193857,-0.784247,0.616476,0.0673647],[-1,-1,-1,0],[0,102,9E+9,9E+9,9E+9,9E+9]];
    PERS robtarget p588:=[[-284.25,-46.11,66.24],[0.0193857,-0.784247,0.616476,0.0673647],[-1,-1,-1,0],[0,102,9E+9,9E+9,9E+9,9E+9]];
    PERS robtarget p590:=[[-284.25,-46.11,66.24],[0.0193857,-0.784247,0.616476,0.0673647],[-1,-1,-1,0],[0,102,9E+9,9E+9,9E+9,9E+9]];
    PERS robtarget p591:=[[-284.25,-46.11,66.24],[0.0193857,-0.784247,0.616476,0.0673647],[-1,-1,-1,0],[0,102,9E+9,9E+9,9E+9,9E+9]];
    PERS robtarget p592:=[[-284.25,-46.11,66.24],[0.0193857,-0.784247,0.616476,0.0673647],[-1,-1,-1,0],[0,102,9E+9,9E+9,9E+9,9E+9]];
    PERS robtarget p593:=[[-284.25,-46.11,66.24],[0.0193857,-0.784247,0.616476,0.0673647],[-1,-1,-1,0],[0,102,9E+9,9E+9,9E+9,9E+9]];
    PERS robtarget mypounce100:=[[18.29,-15.44,503.48],[0.169906,-0.161483,0.329654,0.91454],[-1,0,0,0],[0,-184.719,9E+9,9E+9,9E+9,9E+9]];
    PERS robtarget mypounce150:=[[-650.91,31.30,89.26],[0.116327,-0.124282,0.654165,0.736947],[0,1,0,0],[0,-286.004,9E+9,9E+9,9E+9,9E+9]];
    PERS robtarget p126:=[[-399.05,268.85,394.43],[0.259602,-0.689216,0.461688,0.494401],[-1,-1,1,0],[0,-286.004,9E+9,9E+9,9E+9,9E+9]];
    PERS robtarget p127:=[[-387.38,271.93,393.14],[0.259601,-0.689216,0.461688,0.494401],[-1,-1,1,0],[0,-286.004,9E+9,9E+9,9E+9,9E+9]];
    PERS robtarget p128:=[[-299.50,319.00,366.64],[0.326769,-0.626608,0.575511,0.411549],[0,0,1,0],[0,-286.004,9E+9,9E+9,9E+9,9E+9]];
    PERS robtarget p129:=[[-287.20,311.79,370.99],[0.401395,-0.580915,0.618707,0.344415],[0,0,1,0],[0,-286.004,9E+9,9E+9,9E+9,9E+9]];
    PERS robtarget p251:=[[-131.76,239.79,323.25],[0.659486,-0.28722,0.405018,0.564396],[-1,1,-2,0],[0,-306.3,9E+9,9E+9,9E+9,9E+9]];
    PERS robtarget p261:=[[-131.76,239.79,323.25],[0.659486,-0.28722,0.405018,0.564396],[-1,1,-2,0],[0,-306.3,9E+9,9E+9,9E+9,9E+9]];
    PERS robtarget p200:=[[-154.29,195.35,432.99],[0.323876,-0.134268,0.48472,0.801326],[-1,1,0,0],[0,-184.719,9E+9,9E+9,9E+9,9E+9]];
    PERS robtarget p199:=[[-113.53,150.88,455.82],[0.323876,-0.134268,0.48472,0.801326],[-1,1,0,0],[0,-184.719,9E+9,9E+9,9E+9,9E+9]];
    PERS robtarget mypounce160:=[[-240.26,53.18,506.43],[0.349729,-0.0488935,0.333102,0.874267],[-1,1,0,0],[0,-140.019,9E+9,9E+9,9E+9,9E+9]];
    PERS robtarget p229:=[[-336.78,237.08,417.69],[0.0341496,-0.120948,0.464874,0.876412],[-1,0,0,0],[0,-140.019,9E+9,9E+9,9E+9,9E+9]];
    PERS robtarget p230:=[[-307.13,274.36,383.34],[0.0253369,-0.10342,0.534336,0.838539],[-1,0,0,0],[0,-140.019,9E+9,9E+9,9E+9,9E+9]];
    PERS robtarget mypounce170:=[[-110.25,62.51,506.70],[0.0786297,-0.0971196,0.466016,0.875907],[-1,0,0,0],[0,-56.6292,9E+9,9E+9,9E+9,9E+9]];

    PERS robtarget p262:=[[-479.13,210.77,418.40],[0.376944,-0.165729,0.405226,0.816235],[0,1,0,0],[0,72.809,9E+9,9E+9,9E+9,9E+9]];
    PERS robtarget p263:=[[-389.18,262.86,394.40],[0.376944,-0.165729,0.405226,0.816234],[-1,1,0,0],[0,72.809,9E+9,9E+9,9E+9,9E+9]];
    PERS robtarget p264:=[[-343.21,282.07,383.46],[0.353354,-0.183743,0.524251,0.752689],[-1,1,0,0],[0,72.809,9E+9,9E+9,9E+9,9E+9]];
    PERS robtarget p265:=[[-296.94,314.29,359.80],[0.474107,-0.190787,0.609404,0.606176],[0,1,0,0],[0,72.809,9E+9,9E+9,9E+9,9E+9]];
    PERS robtarget p266:=[[-293.48,315.20,359.78],[0.376606,-0.168654,0.798039,0.439156],[0,0,1,0],[0,72.809,9E+9,9E+9,9E+9,9E+9]];
    PERS robtarget p267:=[[-251.74,310.16,332.74],[0.440559,-0.087755,0.744442,0.493977],[0,1,1,0],[0,72.809,9E+9,9E+9,9E+9,9E+9]];
    PERS robtarget p268:=[[-426.36,161.35,439.18],[0.690968,-0.164283,0.433975,0.554293],[0,2,0,0],[0,72.809,9E+9,9E+9,9E+9,9E+9]];
    PERS robtarget p269:=[[-273.68,277.48,384.52],[0.68121,-0.0999286,0.47362,0.549228],[0,1,0,0],[0,72.809,9E+9,9E+9,9E+9,9E+9]];
    PERS robtarget p270:=[[-228.75,313.10,369.48],[0.530884,-0.0158154,0.558236,0.637404],[0,1,0,0],[0,72.809,9E+9,9E+9,9E+9,9E+9]];
    PERS robtarget p271:=[[-221.87,319.04,354.97],[0.506887,-0.0394596,0.602211,0.615509],[0,1,0,0],[0,72.809,9E+9,9E+9,9E+9,9E+9]];
    PERS robtarget p272:=[[-253.49,316.31,344.31],[0.440559,-0.0877551,0.744442,0.493977],[0,1,1,0],[0,72.809,9E+9,9E+9,9E+9,9E+9]];
    PERS robtarget p273:=[[-251.74,310.16,332.74],[0.440559,-0.087755,0.744442,0.493977],[0,1,1,0],[0,72.809,9E+9,9E+9,9E+9,9E+9]];
    TASK PERS tooldata tool1:=[TRUE,[[0,0,0],[1,0,0,0]],[-1,[0,0,0],[1,0,0,0],0,0,0]];
    CONST robtarget p132:=[[-242.46,206.85,79.24],[0.465919,0.520044,0.567666,0.436152],[0,1,1,0],[0,18.4741,9E+9,9E+9,9E+9,9E+9]];
    PERS robtarget p600:=[[-300.18,30.94,167.83],[0.0758046,0.983318,-0.105712,-0.127137],[0,-1,1,0],[0,-94.382,9E+9,9E+9,9E+9,9E+9]];
    PERS robtarget p601:=[[-312.62,84.28,147.72],[0.0167067,-0.975187,0.117921,0.186618],[0,-1,1,0],[0,-94.382,9E+9,9E+9,9E+9,9E+9]];
    PERS robtarget p602:=[[-305.47,99.90,132.62],[0.0019406,0.973999,-0.0498427,-0.220993],[0,-2,1,0],[0,-94.382,9E+9,9E+9,9E+9,9E+9]];
    PERS robtarget p603:=[[-297.01,140.77,84.43],[0.00194004,0.973999,-0.0498429,-0.220993],[0,-2,1,0],[0,-94.382,9E+9,9E+9,9E+9,9E+9]];
    PERS robtarget p604:=[[-262.46,172.70,44.78],[0.0433988,-0.988115,0.00444524,0.147399],[0,-2,2,0],[0,-94.382,9E+9,9E+9,9E+9,9E+9]];
    PERS robtarget p605:=[[-218.76,182.37,63.41],[0.289259,-0.955005,-0.012675,-0.0642925],[0,-2,2,0],[0,-94.382,9E+9,9E+9,9E+9,9E+9]];
    PERS robtarget p606:=[[-277.68,213.83,330.82],[0.505037,-0.583802,0.585982,0.24645],[-1,-1,0,0],[0,-195,9E+9,9E+9,9E+9,9E+9]];
    PERS robtarget p607:=[[-303.49,216.02,328.89],[0.416767,-0.646308,0.528374,0.359738],[-1,-1,-1,0],[0,-195,9E+9,9E+9,9E+9,9E+9]];
    PERS robtarget p608:=[[-329.18,242.61,321.09],[0.416767,-0.646308,0.528374,0.359738],[-1,-1,-1,0],[0,-195,9E+9,9E+9,9E+9,9E+9]];
    PERS robtarget p609:=[[-22.45,-122.19,118.26],[0.403174,-0.614096,0.639379,0.227004],[-1,-1,0,0],[0,-195,9E+9,9E+9,9E+9,9E+9]];
    PERS robtarget p610:=[[-141.01,71.48,143.52],[0.0361539,-0.996281,-0.0771268,0.0129786],[-1,-2,2,0],[0,-94.382,9E+9,9E+9,9E+9,9E+9]];
    PERS robtarget p611:=[[-164.93,117.75,120.14],[0.0361541,-0.996281,-0.0771268,0.0129786],[0,-2,2,0],[0,-94.382,9E+9,9E+9,9E+9,9E+9]];
    PERS robtarget p612:=[[-191.94,135.66,93.03],[0.036154,-0.996281,-0.0771263,0.0129786],[0,-2,2,0],[0,-94.382,9E+9,9E+9,9E+9,9E+9]];
    PERS robtarget p613:=[[-202.16,155.16,67.69],[0.109149,-0.989499,-0.0899521,-0.0297641],[0,-2,2,0],[0,-94.382,9E+9,9E+9,9E+9,9E+9]];
    PERS robtarget p614:=[[-197.93,170.75,59.56],[0.126656,-0.991052,-0.00590292,-0.0417053],[0,-2,2,0],[0,-94.382,9E+9,9E+9,9E+9,9E+9]];
    PERS robtarget p615:=[[-197.25,180.39,69.56],[0.283507,-0.948467,0.0572129,-0.129465],[0,-1,2,0],[0,-94.382,9E+9,9E+9,9E+9,9E+9]];
    PERS robtarget p616:=[[-277.68,213.83,330.82],[0.505037,-0.583802,0.585982,0.24645],[-1,-1,0,0],[0,-195,9E+9,9E+9,9E+9,9E+9]];
    PERS robtarget p617:=[[-303.49,216.02,328.89],[0.416767,-0.646308,0.528374,0.359738],[-1,-1,-1,0],[0,-195,9E+9,9E+9,9E+9,9E+9]];
    PERS robtarget p618:=[[-329.18,242.61,321.09],[0.416767,-0.646308,0.528374,0.359738],[-1,-1,-1,0],[0,-195,9E+9,9E+9,9E+9,9E+9]];
    PERS robtarget p619:=[[-22.45,-122.19,118.26],[0.403174,-0.614096,0.639379,0.227004],[-1,-1,0,0],[0,-195,9E+9,9E+9,9E+9,9E+9]];
    CONST robtarget mypounce180:=[[-270.02,-132.40,249.19],[0.0106171,0.988751,-0.0899323,-0.119041],[0,-2,1,0],[0,-94.382,9E+9,9E+9,9E+9,9E+9]];
    PERS robtarget p96:=[[-171.05,111.73,122.44],[0.340949,-0.837902,0.394631,-0.16106],[0,-1,2,0],[0,-99.7753,9E+9,9E+9,9E+9,9E+9]];
    PERS robtarget p98:=[[-22.45,-122.19,118.26],[0.403174,-0.614096,0.639379,0.227004],[-1,-1,0,0],[0,-195,9E+9,9E+9,9E+9,9E+9]];
    CONST robtarget mypounce190:=[[44.48,313.16,462.15],[0.441257,-0.541665,0.672728,0.243575],[-1,0,1,0],[0,-286.004,9E+9,9E+9,9E+9,9E+9]];
    CONST robtarget mypounce200:=[[-478.64,264.35,475.85],[0.441257,-0.541665,0.672728,0.243575],[0,0,2,0],[0,-286.004,9E+9,9E+9,9E+9,9E+9]];
    CONST robtarget mypounce210:=[[-548.15,32.82,104.22],[0.441257,-0.541665,0.672727,0.243575],[0,0,2,0],[0,-286.004,9E+9,9E+9,9E+9,9E+9]];
    PERS robtarget p630:=[[-143.32,242.14,414.53],[0.0786299,-0.0971198,0.466016,0.875907],[-1,0,0,0],[0,-56.6292,9E+9,9E+9,9E+9,9E+9]];
    PERS robtarget p631:=[[-195.75,253.59,407.81],[0.0786298,-0.0971197,0.466016,0.875907],[-1,0,0,0],[0,-56.6292,9E+9,9E+9,9E+9,9E+9]];
    PERS robtarget p632:=[[-195.70,253.70,407.60],[0.0674613,-0.0753643,0.572519,0.813628],[-1,0,0,0],[0,-37.6292,9E+9,9E+9,9E+9,9E+9]];
    PERS robtarget p633:=[[-208.21,278.89,396.77],[0.0748337,-0.0896238,0.504416,0.85553],[-1,0,0,0],[0,0.970796,9E+9,9E+9,9E+9,9E+9]];
    PERS robtarget p634:=[[-296.48,298.89,373.93],[0.0806207,-0.101099,0.444846,0.886223],[-1,0,0,0],[0,37.6494,9E+9,9E+9,9E+9,9E+9]];
    PERS robtarget p635:=[[-386.14,251.54,392.71],[0.0847001,-0.109366,0.398979,0.906466],[-1,0,0,0],[0,45.1494,9E+9,9E+9,9E+9,9E+9]];
    PERS robtarget p636:=[[-277.68,213.83,330.82],[0.505037,-0.583802,0.585982,0.24645],[-1,-1,0,0],[0,-195,9E+9,9E+9,9E+9,9E+9]];
    PERS robtarget p637:=[[-303.49,216.02,328.89],[0.416767,-0.646308,0.528374,0.359738],[-1,-1,-1,0],[0,-195,9E+9,9E+9,9E+9,9E+9]];
    PERS robtarget p638:=[[-329.18,242.61,321.09],[0.416767,-0.646308,0.528374,0.359738],[-1,-1,-1,0],[0,-195,9E+9,9E+9,9E+9,9E+9]];
    PERS robtarget p639:=[[-22.45,-122.19,118.26],[0.403174,-0.614096,0.639379,0.227004],[-1,-1,0,0],[0,-195,9E+9,9E+9,9E+9,9E+9]];
    PERS robtarget p640:=[[-198.94,150.86,458.61],[0.0786299,-0.0971198,0.466016,0.875908],[-1,0,0,0],[0,-56.6292,9E+9,9E+9,9E+9,9E+9]];
    PERS robtarget p641:=[[-262.24,163.10,451.28],[0.0786298,-0.09712,0.466016,0.875908],[-1,0,0,0],[0,-56.6292,9E+9,9E+9,9E+9,9E+9]];
    PERS robtarget p642:=[[-242.97,214.35,426.14],[0.0674613,-0.0753643,0.572519,0.813628],[-1,0,0,0],[0,-37.6292,9E+9,9E+9,9E+9,9E+9]];
    PERS robtarget p643:=[[-232.10,243.80,413.67],[0.0748337,-0.0896238,0.504416,0.85553],[-1,0,0,0],[0,0.970796,9E+9,9E+9,9E+9,9E+9]];
    PERS robtarget p644:=[[-329.29,226.68,409.03],[0.0806205,-0.101099,0.444846,0.886223],[-1,0,0,0],[0,37.6494,9E+9,9E+9,9E+9,9E+9]];
    PERS robtarget p645:=[[-393.05,191.76,422.16],[0.0847002,-0.109366,0.398979,0.906466],[-1,0,0,0],[0,45.1494,9E+9,9E+9,9E+9,9E+9]];
    PERS robtarget p646:=[[-277.68,213.83,330.82],[0.505037,-0.583802,0.585982,0.24645],[-1,-1,0,0],[0,-195,9E+9,9E+9,9E+9,9E+9]];
    PERS robtarget p647:=[[-303.49,216.02,328.89],[0.416767,-0.646308,0.528374,0.359738],[-1,-1,-1,0],[0,-195,9E+9,9E+9,9E+9,9E+9]];
    PERS robtarget p648:=[[-329.18,242.61,321.09],[0.416767,-0.646308,0.528374,0.359738],[-1,-1,-1,0],[0,-195,9E+9,9E+9,9E+9,9E+9]];
    PERS robtarget p649:=[[-22.45,-122.19,118.26],[0.403174,-0.614096,0.639379,0.227004],[-1,-1,0,0],[0,-195,9E+9,9E+9,9E+9,9E+9]];
    PERS robtarget mypounce220:=[[-553.13,109.86,493.22],[0.0752025,-0.109552,0.474601,0.870113],[-1,0,0,0],[0,72.809,9E+9,9E+9,9E+9,9E+9]];
    PERS robtarget mypounce230:=[[2.89,50.89,504.75],[0.585257,-0.478952,0.469777,0.455399],[-1,1,0,0],[0,72.809,9E+9,9E+9,9E+9,9E+9]];
    PERS robtarget mypounce240:=[[-568.28,-124.52,-146.95],[0.150555,-0.0794425,0.859081,0.482703],[0,1,0,0],[0,62.0225,9E+9,9E+9,9E+9,9E+9]];
    PERS robtarget mypounce250:=[[227.24,-296.81,-41.89],[0.450262,-0.587835,0.630347,0.233186],[-1,-1,2,0],[0,30.1629,9E+9,9E+9,9E+9,9E+9]];
    PERS robtarget checkp1:=[[-49.48,55.23,198.94],[0.456001,-0.656027,0.531792,0.28087],[-1,-1,2,0],[0,0.0198783,9E+9,9E+9,9E+9,9E+9]];
    PERS robtarget checkp11:=[[-80.29,252.73,451.21],[0.456001,-0.656027,0.531792,0.28087],[-1,-1,2,0],[0,0.0198783,9E+9,9E+9,9E+9,9E+9]];
    PERS robtarget checkp21:=[[-152.64,34.52,72.71],[0.456001,-0.656027,0.531792,0.28087],[0,-1,2,0],[0,67.5,9E+9,9E+9,9E+9,9E+9]];
    PERS wobjdata wobj2:=[FALSE,TRUE,"",[[0,0,0],[1,0,0,0]],[[0,0,0],[1,0,0,0]]];



    !*************************************************************************************

    PROC Main()
	    !0464 Vane3\
        currentTool:= Cascade_175mm;
        !wobj is zeroed
        currentWorkObject:=wobj1;
        !MoveAbsJ [[0,0,0,0,0,0],[0,0,9E+9,9E+9,9E+9,9E+9]]\NoEOffs, v1000, z50, currentTool\WObj:=currentWorkObject;
        !MoveJ checkp1, v100, fine, currentTool\WObj:=currentWorkObject;
        !MoveJ checkp11, v100, fine, currentTool\WObj:=currentWorkObject;
        !MoveJ checkp21, v100, fine, currentTool\WObj:=currentWorkObject;

        TPErase;
        !prompt operator
        TPWrite "When Ready press 'Operator Start'";
        WaitDI DI_OP_Start, 1;
        TPErase;

        ! move to home position
        MoveL home30, v400, z10, currentTool\WObj:=currentWorkObject;

        ! get part program from operator
        itemSelected:=UIListView(\Result:=buttonAnswer,\Header:="FSNH_0464",partProgram,\Buttons:=btnOKCancel,\Icon:=iconInfo,\DefaultIndex:=1);

        IF buttonAnswer=resOK THEN
            IF itemSelected=1 THEN
              topCoat;
            ELSEIF itemSelected=2 THEN
              flashCoat;
            ELSE
              GOTO StopCycle;
            ENDIF
        ELSE
            ! if user selects cancel then stop cycle
            GOTO StopCycle;
        ENDIF


        StopCycle:
        MoveL home30, v400, z10, currentTool\WObj:=currentWorkObject;

    ENDPROC


    PROC topCoat()
        currentTool:= Cascade_175mm;
	    ! set cycle counters
        coatingCycleCounter:=5;
        TPReadNum reg7, "how many heat passes?";

        ! allow operator to change the number of coating cycles from the default value
        defaultValueString := "default value = " + NumtoStr(coatingCycleCounter,0);
        coatingCycleCounter := UINumEntry (\Header:="Change Coating Cycles", \MsgArray:=["How many coating cycles?", defaultValueString], \InitValue:=coatingCycleCounter, \AsInteger);

        ! move to pounce position
        MoveJ home30, v800, z10, currentTool\WObj:=currentWorkObject;
        TPErase;
        TPWrite "Start Gun, and press 'Cycle Start' to Start";

        WaitDI DI_OP_start, 1;
        TPErase;
        !heat passes
        IF reg7 > 0 THEN
            WHILE reg7>0 DO
                !sprays 3 sections fo platform
                PLATFORM;
                !sprays airfoils
                CVAirfoil1;
                Airfoilinner1;
                !sprays last platform section
                PL4;
                !continues with airfoil
                AirfoilCCOuter;
                Airlfoilinner2;
                !sprays the whole shroud
                SHROUD;

              MoveL home30, v800, z10, currentTool\WObj:=currentWorkObject;

              ! decrement the cycle counter
              reg7:=reg7-1;
              TPErase;
              TPWrite "number of coating cycles remaining = "\Num:=reg7;
              !
            ENDWHILE
        ENDIF

        MoveJ home30, v800, z10, currentTool\WObj:=currentWorkObject;
        !turn powder on
        TPWrite "Turn on powder, and press 'Cycle Start' to Start";
        !
        WaitDI DI_OP_start, 1;
        TPErase;
        MoveL home30, v800, z10, currentTool\WObj:=currentWorkObject;

        WHILE coatingCycleCounter>0 DO
            !sprays 3 sections fo platform
            PLATFORM;
            !sprays airfoils
            CVAirfoil1;
            Airfoilinner1;
            !sprays last platform section
            PL4;
            !continues with airfoil
            AirfoilCCOuter;
            Airlfoilinner2;
            !sprays the whole shroud
            SHROUD;

          MoveL home30, v800, z10, currentTool\WObj:=currentWorkObject;

          ! decrement the cycle counter
          coatingCycleCounter:=coatingCycleCounter-1;
          TPErase;
          TPWrite "number of coating cycles remaining = "\Num:=coatingCycleCounter;
          !
        ENDWHILE
        !
        SKIP:
        !
        ! move to home position
        MoveL home30, v800, z10, currentTool\WObj:=currentWorkObject;

    ENDPROC

    !*************************************************************************************

     PROC flashCoat()
         currentTool:= Cascade_175mm;
		 ! set cycle counters
        coatingCycleCounter:=5;
        TPReadNum reg7, "how many heat passes?";

        ! allow operator to change the number of coating cycles from the default value
        defaultValueString := "default value = " + NumtoStr(coatingCycleCounter,0);
        coatingCycleCounter := UINumEntry (\Header:="Change Coating Cycles", \MsgArray:=["How many coating cycles?", defaultValueString], \InitValue:=coatingCycleCounter, \AsInteger);

        ! move to pounce position
        MoveJ home30, v800, z10, currentTool\WObj:=currentWorkObject;
        TPErase;
        TPWrite "Start Gun, and press 'Cycle Start' to Start";

        WaitDI DI_OP_start, 1;
        TPErase;
        !heat passes
        IF reg7 > 0 THEN
            WHILE reg7>0 DO
                !sprays 3 sections fo platform
                PLATFORM;
                !sprays airfoils
                CVAirfoil1;
                Airfoilinner1;
                !sprays last platform section
                PL4;
                !continues with airfoil
                AirfoilCCOuter;
                Airlfoilinner2;
                !sprays the whole shroud
                SHROUD;

              MoveL home30, v800, z10, currentTool\WObj:=currentWorkObject;

              ! decrement the cycle counter
              reg7:=reg7-1;
              TPErase;
              TPWrite "number of coating cycles remaining = "\Num:=reg7;
              !
            ENDWHILE
        ENDIF

        MoveJ home30, v800, z10, currentTool\WObj:=currentWorkObject;
        !turn powder on
        TPWrite "Turn on powder, and press 'Cycle Start' to Start";
        !
        WaitDI DI_OP_start, 1;
        TPErase;
        MoveL home30, v800, z10, currentTool\WObj:=currentWorkObject;

        WHILE coatingCycleCounter>0 DO
            !sprays 3 sections fo platform
            PLATFORM;
            !sprays airfoils
            CVAirfoil1;
            Airfoilinner1;
            !sprays last platform section
            PL4;
            !continues with airfoil
            AirfoilCCOuter;
            Airlfoilinner2;
            !sprays the whole shroud
            SHROUD;

          MoveL home30, v800, z10, currentTool\WObj:=currentWorkObject;

          ! decrement the cycle counter
          coatingCycleCounter:=coatingCycleCounter-1;
          TPErase;
          TPWrite "number of coating cycles remaining = "\Num:=coatingCycleCounter;
          !
        ENDWHILE
        !
        SKIP:
        !
        ! move to home position
        MoveL home30, v800, z10, currentTool\WObj:=currentWorkObject;
        RETURN;
    ENDPROC

    !***********************************************************************************************************!


    PROC AIRFOIL()
        !sprays airfoil
        CVAirfoil1;
        Airfoilinner1;
        AirfoilCCOuter;
        Airlfoilinner2;

    ENDPROC

    PROC SHROUD()
        !
        !Shroud1;
        MoveL mypounce150, v1000, z50, currentTool\WObj:=currentWorkObject;
		MoveL mypounce70, v1000, z50, currentTool\WObj:=currentWorkObject;
		MoveL mypounce100, v1000, z50, currentTool\WObj:=currentWorkObject;

        SpeedFactors_3 3,3,3,3,3,3,3,3,3,3;
        SpeedFactors_4 3,3,3,3,3,3,3,3,3,3;
        Para4 7,500,199,208,6;

        !shroud2;
        MoveL mypounce160, v1000, z50, currentTool\WObj:=currentWorkObject;

        SpeedFactors_3 3,3,3,3,3,3,3,3,3,3;
        SpeedFactors_4 3,3,3,3,3,3,3,3,3,3;
        Para4 7,500,221,229,5;

        !Shroud3;
        MoveL mypounce170, v1000, z50, currentTool\WObj:=currentWorkObject;

        SpeedFactors_3 3,3,3,3,3,3,3,3,3,3;
        SpeedFactors_4 3,3,3,3,3,3,3,3,3,3;
        Para4 7,500,630,640,6;

        !Shroud4;
        MoveL mypounce220, v1000, z50, currentTool\WObj:=currentWorkObject;

        SpeedFactors_3 3,3,3,3,3,3,3,3,3,3;
        SpeedFactors_4 3,3,3,3,3,3,3,3,3,3;
        Para4 7,500,262,268,5;
		MoveL mypounce240, v1000, z50, currentTool\WObj:=currentWorkObject;
		MoveL mypounce250, v1000, z50, currentTool\WObj:=currentWorkObject;

        RETURN;
        MoveL p199, v500, z1, currentTool\WObj:=currentWorkObject;
        MoveL p200, v500, z1, currentTool\WObj:=currentWorkObject;
        MoveL p201, v500, z1, currentTool\WObj:=currentWorkObject;
        MoveL p202, v500, z1, currentTool\WObj:=currentWorkObject;
		MoveL p203, v500, z1, currentTool\WObj:=currentWorkObject;
		MoveL p204, v500, z1, currentTool\WObj:=currentWorkObject;
		!MoveL p205, v500, z1, currentTool\WObj:=currentWorkObject;
		!MoveL p206, v500, z1, currentTool\WObj:=currentWorkObject;
		!MoveL p207, v500, z1, currentTool\WObj:=currentWorkObject;

        MoveL p208, v500, z1, currentTool\WObj:=currentWorkObject;
		MoveL p209, v500, z1, currentTool\WObj:=currentWorkObject;
		MoveL p210, v500, z1, currentTool\WObj:=currentWorkObject;
		MoveL p211, v500, z1, currentTool\WObj:=currentWorkObject;
		MoveL p212, v500, z1, currentTool\WObj:=currentWorkObject;
        MoveL p213, v500, z1, currentTool\WObj:=currentWorkObject;

        !shroud2
        !MoveL p220, v500, z1, currentTool\WObj:=currentWorkObject;
        MoveL p221, v500, z1, currentTool\WObj:=currentWorkObject;
        MoveL p222, v500, z1, currentTool\WObj:=currentWorkObject;
        MoveL p223, v500, z1, currentTool\WObj:=currentWorkObject;
		MoveL p224, v500, z1, currentTool\WObj:=currentWorkObject;
		MoveL p225, v500, z1, currentTool\WObj:=currentWorkObject;
		!MoveL p226, v500, z1, currentTool\WObj:=currentWorkObject;
		!MoveL p227, v500, z1, currentTool\WObj:=currentWorkObject;
		!MoveL p228, v500, z1, currentTool\WObj:=currentWorkObject;

        MoveL p229, v500, z1, currentTool\WObj:=currentWorkObject;
		MoveL p230, v500, z1, currentTool\WObj:=currentWorkObject;
		MoveL p231, v500, z1, currentTool\WObj:=currentWorkObject;
		MoveL p232, v500, z1, currentTool\WObj:=currentWorkObject;
		MoveL p233, v500, z1, currentTool\WObj:=currentWorkObject;
        !MoveL p234, v500, z1, currentTool\WObj:=currentWorkObject;
        !MoveL p235, v500, z1, currentTool\WObj:=currentWorkObject;

        !Shroud 3
         MoveL p630, v500, z1, currentTool\WObj:=currentWorkObject;
        MoveL p631, v500, z1, currentTool\WObj:=currentWorkObject;
        MoveL p632, v500, z1, currentTool\WObj:=currentWorkObject;
        MoveL p633, v500, z1, currentTool\WObj:=currentWorkObject;
		MoveL p634, v500, z1, currentTool\WObj:=currentWorkObject;
		MoveL p635, v500, z1, currentTool\WObj:=currentWorkObject;
        !MoveL p636, v500, z1, currentTool\WObj:=currentWorkObject;
		!MoveL p637, v500, z1, currentTool\WObj:=currentWorkObject;
		!MoveL p638, v500, z1, currentTool\WObj:=currentWorkObject;
        !MoveL p639, v500, z1, currentTool\WObj:=currentWorkObject;

        MoveL p640, v500, z1, currentTool\WObj:=currentWorkObject;
        MoveL p641, v500, z1, currentTool\WObj:=currentWorkObject;
        MoveL p642, v500, z1, currentTool\WObj:=currentWorkObject;
        MoveL p643, v500, z1, currentTool\WObj:=currentWorkObject;
		MoveL p644, v500, z1, currentTool\WObj:=currentWorkObject;
		MoveL p645, v500, z1, currentTool\WObj:=currentWorkObject;
		!MoveL p646, v500, z1, currentTool\WObj:=currentWorkObject;
		!MoveL p647, v500, z1, currentTool\WObj:=currentWorkObject;
		!MoveL p648, v500, z1, currentTool\WObj:=currentWorkObject;
        !MoveL p649, v500, z1, currentTool\WObj:=currentWorkObject;

        !shroud 4
        MoveL p262, v500, z1, currentTool\WObj:=currentWorkObject;
        MoveL p263, v500, z1, currentTool\WObj:=currentWorkObject;
        MoveL p264, v500, z1, currentTool\WObj:=currentWorkObject;
        MoveL p265, v500, z1, currentTool\WObj:=currentWorkObject;
		MoveL p266, v500, z1, currentTool\WObj:=currentWorkObject;
		!MoveL p267, v500, z1, currentTool\WObj:=currentWorkObject;

        MoveL p268, v500, z1, currentTool\WObj:=currentWorkObject;
		MoveL p269, v500, z1, currentTool\WObj:=currentWorkObject;
		MoveL p270, v500, z1, currentTool\WObj:=currentWorkObject;
        MoveL p271, v500, z1, currentTool\WObj:=currentWorkObject;
		MoveL p272, v500, z1, currentTool\WObj:=currentWorkObject;
		!MoveL p273, v500, z1, currentTool\WObj:=currentWorkObject;

    ENDPROC



    PROC PLATFORM()

        !PL1;
        MoveL mypounce10, v1000, z50, currentTool\WObj:=currentWorkObject;
        SpeedFactors_3 3,3,3,3,3,3,3,3,3,3;
        SpeedFactors_4 3,3,3,3,3,3,3,3,3,3;

        Para4 8,500,19,26,6;

        !PL2;
        MoveL mypounce, v1000, z50, currentTool\WObj:=currentWorkObject;
        SpeedFactors_3 3,3,3,3,3,3,3,3,3,3;
        SpeedFactors_4 3,3,3,3,3,3,3,3,3,3;

        Para4 8,500,1,8,6;

        !PL3;
        MoveL mypounce20, v1000, z50, currentTool\WObj:=currentWorkObject;
        SpeedFactors_3 3,3,3,3,3,3,3,3,3,3;
        SpeedFactors_4 3,3,3,3,3,3,3,3,3,3;

        Para4 8,500,40,48,7;

        RETURN;
        !PL1
        MoveL p19, v1000, z50, currentTool\WObj:=currentWorkObject;
        MoveL p20, v1000, z50, currentTool\WObj:=currentWorkObject;
		MoveL p21, v500, z1, currentTool\WObj:=currentWorkObject;
		MoveL p22, v500, z1, currentTool\WObj:=currentWorkObject;
		MoveL p23, v500, z1, currentTool\WObj:=currentWorkObject;
		MoveL p24, v500, z1, currentTool\WObj:=currentWorkObject;
		MoveL p25, v500, z1, currentTool\WObj:=currentWorkObject;

        MoveL p26, v500, z1, currentTool\WObj:=currentWorkObject;
		MoveL p27, v500, z1, currentTool\WObj:=currentWorkObject;
		MoveL p28, v500, z1, currentTool\WObj:=currentWorkObject;
		MoveL p29, v500, z1, currentTool\WObj:=currentWorkObject;
        MoveL p30, v500, z1, currentTool\WObj:=currentWorkObject;
        MoveL p31, v500, z1, currentTool\WObj:=currentWorkObject;

        !PL2
        MoveL p1, v1000, z50, currentTool\WObj:=currentWorkObject;
		MoveL p2, v500, z1, currentTool\WObj:=currentWorkObject;
		MoveL p3, v500, z1, currentTool\WObj:=currentWorkObject;
		MoveL p4, v500, z1, currentTool\WObj:=currentWorkObject;
		MoveL p5, v500, z1, currentTool\WObj:=currentWorkObject;
		MoveL p6, v500, z1, currentTool\WObj:=currentWorkObject;
		!MoveL p7, v500, z1, currentTool\WObj:=currentWorkObject;

		MoveL p8, v500, z1, currentTool\WObj:=currentWorkObject;
		MoveL p9, v500, z1, currentTool\WObj:=currentWorkObject;
		MoveL p10, v500, z1, currentTool\WObj:=currentWorkObject;
        MoveL p11, v500, z1, currentTool\WObj:=currentWorkObject;
        MoveL p12, v500, z1, currentTool\WObj:=currentWorkObject;
        MoveL p13, v500, z1, currentTool\WObj:=currentWorkObject;

        !PL3
        MoveL p40, v1000, z50, currentTool\WObj:=currentWorkObject;
        MoveL p41, v1000, z50, currentTool\WObj:=currentWorkObject;
		MoveL p42, v500, z1, currentTool\WObj:=currentWorkObject;
		MoveL p43, v500, z1, currentTool\WObj:=currentWorkObject;
		MoveL p44, v500, z1, currentTool\WObj:=currentWorkObject;
		MoveL p45, v500, z1, currentTool\WObj:=currentWorkObject;
		MoveL p46, v500, z1, currentTool\WObj:=currentWorkObject;

		MoveL p48, v500, z1, currentTool\WObj:=currentWorkObject;
		MoveL p49, v500, z1, currentTool\WObj:=currentWorkObject;
		MoveL p50, v500, z1, currentTool\WObj:=currentWorkObject;
        MoveL p51, v500, z1, currentTool\WObj:=currentWorkObject;
        MoveL p52, v500, z1, currentTool\WObj:=currentWorkObject;
        MoveL p53, v500, z1, currentTool\WObj:=currentWorkObject;
        MoveL p54, v500, z1, currentTool\WObj:=currentWorkObject;
    ENDPROC


	PROC PL1()
        MoveL mypounce10, v1000, z50, currentTool\WObj:=currentWorkObject;
        SpeedFactors_3 3,3,3,3,3,3,3,3,3,3;
        SpeedFactors_4 3,3,3,3,3,3,3,3,3,3;

        Para4 8,500,19,26,6;

        RETURN;
        MoveL p19, v1000, z50, currentTool\WObj:=currentWorkObject;
        MoveL p20, v1000, z50, currentTool\WObj:=currentWorkObject;
		MoveL p21, v500, z1, currentTool\WObj:=currentWorkObject;
		MoveL p22, v500, z1, currentTool\WObj:=currentWorkObject;
		MoveL p23, v500, z1, currentTool\WObj:=currentWorkObject;
		MoveL p24, v500, z1, currentTool\WObj:=currentWorkObject;
		MoveL p25, v500, z1, currentTool\WObj:=currentWorkObject;

        MoveL p26, v500, z1, currentTool\WObj:=currentWorkObject;
		MoveL p27, v500, z1, currentTool\WObj:=currentWorkObject;
		MoveL p28, v500, z1, currentTool\WObj:=currentWorkObject;
		MoveL p29, v500, z1, currentTool\WObj:=currentWorkObject;
        MoveL p30, v500, z1, currentTool\WObj:=currentWorkObject;
        MoveL p31, v500, z1, currentTool\WObj:=currentWorkObject;
	ENDPROC
	PROC PL2()
        !inner platform
		MoveL mypounce, v1000, z50, currentTool\WObj:=currentWorkObject;
        SpeedFactors_3 3,3,3,3,3,3,3,3,3,3;
        SpeedFactors_4 3,3,3,3,3,3,3,3,3,3;

        Para4 8,500,1,8,6;

        RETURN;
        MoveL p1, v1000, z50, currentTool\WObj:=currentWorkObject;
		MoveL p2, v500, z1, currentTool\WObj:=currentWorkObject;
		MoveL p3, v500, z1, currentTool\WObj:=currentWorkObject;
		MoveL p4, v500, z1, currentTool\WObj:=currentWorkObject;
		MoveL p5, v500, z1, currentTool\WObj:=currentWorkObject;
		MoveL p6, v500, z1, currentTool\WObj:=currentWorkObject;
		!MoveL p7, v500, z1, currentTool\WObj:=currentWorkObject;

		MoveL p8, v500, z1, currentTool\WObj:=currentWorkObject;
		MoveL p9, v500, z1, currentTool\WObj:=currentWorkObject;
		MoveL p10, v500, z1, currentTool\WObj:=currentWorkObject;
        MoveL p11, v500, z1, currentTool\WObj:=currentWorkObject;
        MoveL p12, v500, z1, currentTool\WObj:=currentWorkObject;
        MoveL p13, v500, z1, currentTool\WObj:=currentWorkObject;
	ENDPROC
	PROC PL3()

		MoveL mypounce20, v1000, z50, currentTool\WObj:=currentWorkObject;
        SpeedFactors_3 3,3,3,3,3,3,3,3,3,3;
        SpeedFactors_4 3,3,3,3,3,3,3,3,3,3;

        Para4 8,500,40,48,7;

        RETURN;

        MoveL p40, v1000, z50, currentTool\WObj:=currentWorkObject;
        MoveL p41, v1000, z50, currentTool\WObj:=currentWorkObject;
		MoveL p42, v500, z1, currentTool\WObj:=currentWorkObject;
		MoveL p43, v500, z1, currentTool\WObj:=currentWorkObject;
		MoveL p44, v500, z1, currentTool\WObj:=currentWorkObject;
		MoveL p45, v500, z1, currentTool\WObj:=currentWorkObject;
		MoveL p46, v500, z1, currentTool\WObj:=currentWorkObject;


		MoveL p48, v500, z1, currentTool\WObj:=currentWorkObject;
		MoveL p49, v500, z1, currentTool\WObj:=currentWorkObject;
		MoveL p50, v500, z1, currentTool\WObj:=currentWorkObject;
        MoveL p51, v500, z1, currentTool\WObj:=currentWorkObject;
        MoveL p52, v500, z1, currentTool\WObj:=currentWorkObject;
        MoveL p53, v500, z1, currentTool\WObj:=currentWorkObject;
        MoveL p54, v500, z1, currentTool\WObj:=currentWorkObject;
	ENDPROC

    PROC PL4()
		MoveL mypounce180, v1000, z50, currentTool\WObj:=currentWorkObject;
        SpeedFactors_3 3,3,3,3,3,3,3,3,3,3;
        SpeedFactors_4 3,3,3,3,3,3,3,3,3,3;

        Para4 8,500,600,610,6;

        RETURN;
        MoveL p600, v500, z1, currentTool\WObj:=currentWorkObject;
        MoveL p601, v500, z1, currentTool\WObj:=currentWorkObject;
		MoveL p602, v500, z1, currentTool\WObj:=currentWorkObject;
		MoveL p603, v500, z1, currentTool\WObj:=currentWorkObject;
		MoveL p604, v500, z1, currentTool\WObj:=currentWorkObject;
		MoveL p605, v500, z1, currentTool\WObj:=currentWorkObject;
		!MoveL p606, v500, z1, currentTool\WObj:=currentWorkObject;
        !MoveL p607, v500, z1, currentTool\WObj:=currentWorkObject;
		!MoveL p608, v500, z1, currentTool\WObj:=currentWorkObject;
		!MoveL p609, v500, z1, currentTool\WObj:=currentWorkObject;

        MoveL p610, v500, z1, currentTool\WObj:=currentWorkObject;
		MoveL p611, v500, z1, currentTool\WObj:=currentWorkObject;
        MoveL p612, v500, z1, currentTool\WObj:=currentWorkObject;
        MoveL p613, v500, z1, currentTool\WObj:=currentWorkObject;
        MoveL p614, v500, z1, currentTool\WObj:=currentWorkObject;
		MoveL p615, v500, z1, currentTool\WObj:=currentWorkObject;
        !MoveL p616, v500, z1, currentTool\WObj:=currentWorkObject;
        !MoveL p617, v500, z1, currentTool\WObj:=currentWorkObject;
        !MoveL p618, v500, z1, currentTool\WObj:=currentWorkObject;
		!MoveL p619, v500, z1, currentTool\WObj:=currentWorkObject;


	ENDPROC


    PROC CVAirfoil1()
        MoveL mypounce30, v1000, z50, currentTool\WObj:=currentWorkObject;

        SpeedFactors_3 2,2,1,1,1,2,2,2,2,2;
        SpeedFactors_4 2,2,1,1,1,2,2,2,2,2;

        Para4 8,500,60,67,7;

        RETURN;
        MoveL p60, v500, z1, currentTool\WObj:=currentWorkObject;
        MoveL p61, v500, z1, currentTool\WObj:=currentWorkObject;
		MoveL p62, v500, z1, currentTool\WObj:=currentWorkObject;
		MoveL p63, v500, z1, currentTool\WObj:=currentWorkObject;
		MoveL p64, v500, z1, currentTool\WObj:=currentWorkObject;
		MoveL p65, v500, z1, currentTool\WObj:=currentWorkObject;
		MoveL p66, v500, z1, currentTool\WObj:=currentWorkObject;


		MoveL p67, v500, z1, currentTool\WObj:=currentWorkObject;
		MoveL p68, v500, z1, currentTool\WObj:=currentWorkObject;
		MoveL p69, v500, z1, currentTool\WObj:=currentWorkObject;
        MoveL p70, v500, z1, currentTool\WObj:=currentWorkObject;
        MoveL p71, v500, z1, currentTool\WObj:=currentWorkObject;
        MoveL p72, v500, z1, currentTool\WObj:=currentWorkObject;
        MoveL p73, v500, z1, currentTool\WObj:=currentWorkObject;

		ENDPROC

	PROC Airfoilinner1()
        MoveL mypounce40, v1000, z50, currentTool\WObj:=currentWorkObject;
        SpeedFactors_3 1,3,3,1,1,1,1,1,1,1;
        SpeedFactors_4 1,3,3,1,1,1,1,1,1,1;

        Para4 8,500,80,89,9;

        RETURN;
        MoveL p80, v500, z1, currentTool\WObj:=currentWorkObject;
        MoveL p81, v500, z1, currentTool\WObj:=currentWorkObject;
		MoveL p82, v500, z1, currentTool\WObj:=currentWorkObject;
		MoveL p83, v500, z1, currentTool\WObj:=currentWorkObject;
		MoveL p84, v500, z1, currentTool\WObj:=currentWorkObject;
		MoveL p85, v500, z1, currentTool\WObj:=currentWorkObject;
		MoveL p86, v500, z1, currentTool\WObj:=currentWorkObject;
		MoveL p87, v500, z1, currentTool\WObj:=currentWorkObject;
		MoveL p88, v500, z1, currentTool\WObj:=currentWorkObject;

        MoveL p89, v500, z1, currentTool\WObj:=currentWorkObject;
		MoveL p90, v500, z1, currentTool\WObj:=currentWorkObject;
		MoveL p91, v500, z1, currentTool\WObj:=currentWorkObject;
        MoveL p92, v500, z1, currentTool\WObj:=currentWorkObject;
        MoveL p93, v500, z1, currentTool\WObj:=currentWorkObject;
        MoveL p94, v500, z1, currentTool\WObj:=currentWorkObject;
		MoveL p95, v500, z1, currentTool\WObj:=currentWorkObject;
		MoveL p96, v500, z1, currentTool\WObj:=currentWorkObject;
        MoveL p97, v500, z1, currentTool\WObj:=currentWorkObject;
        !MoveL p98, v500, z1, currentTool\WObj:=currentWorkObject;

		ENDPROC
	PROC AirfoilCCOuter()
        MoveL mypounce50, v1000, z50, currentTool\WObj:=currentWorkObject;
        SpeedFactors_3 3,3,3,3,3,3,3,3,3,3;
        SpeedFactors_4 3,3,3,3,3,3,3,3,3,3;

        Para4 8,500,100,107,6;

        RETURN;
        MoveL p100, v500, z1, currentTool\WObj:=currentWorkObject;
        MoveL p101, v500, z1, currentTool\WObj:=currentWorkObject;
		MoveL p102, v500, z1, currentTool\WObj:=currentWorkObject;
		MoveL p103, v500, z1, currentTool\WObj:=currentWorkObject;
		MoveL p104, v500, z1, currentTool\WObj:=currentWorkObject;
		MoveL p105, v500, z1, currentTool\WObj:=currentWorkObject;
		!MoveL p106, v500, z1, currentTool\WObj:=currentWorkObject;

        MoveL p107, v500, z1, currentTool\WObj:=currentWorkObject;
		MoveL p108, v500, z1, currentTool\WObj:=currentWorkObject;
		MoveL p109, v500, z1, currentTool\WObj:=currentWorkObject;
		MoveL p110, v500, z1, currentTool\WObj:=currentWorkObject;
		MoveL p111, v500, z1, currentTool\WObj:=currentWorkObject;
        MoveL p112, v500, z1, currentTool\WObj:=currentWorkObject;
        !MoveL p113, v500, z1, currentTool\WObj:=currentWorkObject;
		ENDPROC
	PROC Airlfoilinner2()
		MoveL mypounce60, v1000, z50, currentTool\WObj:=currentWorkObject;
		MoveL mypounce190, v1000, z50, currentTool\WObj:=currentWorkObject;
		MoveL mypounce200, v1000, z50, currentTool\WObj:=currentWorkObject;
		MoveL mypounce210, v1000, z50, currentTool\WObj:=currentWorkObject;
        SpeedFactors_3 3,3,3,3,3,3,3,3,3,3;
        SpeedFactors_4 3,3,3,3,3,3,3,3,3,3;

        Para4 8, 500, 120, 126, 4;

        RETURN;
        MoveL p120, v500, z1, currentTool\WObj:=currentWorkObject;
        MoveL p121, v500, z1, currentTool\WObj:=currentWorkObject;
		MoveL p122, v500, z1, currentTool\WObj:=currentWorkObject;
		MoveL p123, v500, z1, currentTool\WObj:=currentWorkObject;
		!MoveL p104, v500, z1, currentTool\WObj:=currentWorkObject;
		!MoveL p105, v500, z1, currentTool\WObj:=currentWorkObject;
		!MoveL p106, v500, z1, currentTool\WObj:=currentWorkObject;

        MoveL p126, v500, z1, currentTool\WObj:=currentWorkObject;
		MoveL p127, v500, z1, currentTool\WObj:=currentWorkObject;
		MoveL p128, v500, z1, currentTool\WObj:=currentWorkObject;
		MoveL p129, v500, z1, currentTool\WObj:=currentWorkObject;
		!MoveL p111, v500, z1, currentTool\WObj:=currentWorkObject;
        !MoveL p112, v500, z1, currentTool\WObj:=currentWorkObject;
        !MoveL p113, v500, z1, currentTool\WObj:=currentWorkObject;

	ENDPROC
	PROC Shroud1()
		MoveL mypounce150, v1000, z50, currentTool\WObj:=currentWorkObject;
		MoveL mypounce70, v1000, z50, currentTool\WObj:=currentWorkObject;
		MoveL mypounce100, v1000, z50, currentTool\WObj:=currentWorkObject;

        SpeedFactors_3 3,3,3,3,3,3,3,3,3,3;
        SpeedFactors_4 3,3,3,3,3,3,3,3,3,3;
        Para4 7,500,199,208,6;

        RETURN;
        MoveL p199, v500, z1, currentTool\WObj:=currentWorkObject;
        MoveL p200, v500, z1, currentTool\WObj:=currentWorkObject;
        MoveL p201, v500, z1, currentTool\WObj:=currentWorkObject;
        MoveL p202, v500, z1, currentTool\WObj:=currentWorkObject;
		MoveL p203, v500, z1, currentTool\WObj:=currentWorkObject;
		MoveL p204, v500, z1, currentTool\WObj:=currentWorkObject;
		!MoveL p205, v500, z1, currentTool\WObj:=currentWorkObject;
		!MoveL p206, v500, z1, currentTool\WObj:=currentWorkObject;
		!MoveL p207, v500, z1, currentTool\WObj:=currentWorkObject;

        MoveL p208, v500, z1, currentTool\WObj:=currentWorkObject;
		MoveL p209, v500, z1, currentTool\WObj:=currentWorkObject;
		MoveL p210, v500, z1, currentTool\WObj:=currentWorkObject;
		MoveL p211, v500, z1, currentTool\WObj:=currentWorkObject;
		MoveL p212, v500, z1, currentTool\WObj:=currentWorkObject;
        MoveL p213, v500, z1, currentTool\WObj:=currentWorkObject;



	ENDPROC


	PROC shroud2()
		MoveL mypounce160, v1000, z50, currentTool\WObj:=currentWorkObject;

        SpeedFactors_3 3,3,3,3,3,3,3,3,3,3;
        SpeedFactors_4 3,3,3,3,3,3,3,3,3,3;
        Para4 7,500,221,229,5;

        RETURN;
        !MoveL p220, v500, z1, currentTool\WObj:=currentWorkObject;
        MoveL p221, v500, z1, currentTool\WObj:=currentWorkObject;
        MoveL p222, v500, z1, currentTool\WObj:=currentWorkObject;
        MoveL p223, v500, z1, currentTool\WObj:=currentWorkObject;
		MoveL p224, v500, z1, currentTool\WObj:=currentWorkObject;
		MoveL p225, v500, z1, currentTool\WObj:=currentWorkObject;
		!MoveL p226, v500, z1, currentTool\WObj:=currentWorkObject;
		!MoveL p227, v500, z1, currentTool\WObj:=currentWorkObject;
		!MoveL p228, v500, z1, currentTool\WObj:=currentWorkObject;

        MoveL p229, v500, z1, currentTool\WObj:=currentWorkObject;
		MoveL p230, v500, z1, currentTool\WObj:=currentWorkObject;
		MoveL p231, v500, z1, currentTool\WObj:=currentWorkObject;
		MoveL p232, v500, z1, currentTool\WObj:=currentWorkObject;
		MoveL p233, v500, z1, currentTool\WObj:=currentWorkObject;
        !MoveL p234, v500, z1, currentTool\WObj:=currentWorkObject;
        !MoveL p235, v500, z1, currentTool\WObj:=currentWorkObject;

	ENDPROC
	PROC Shroud3()
		MoveL mypounce170, v1000, z50, currentTool\WObj:=currentWorkObject;

        SpeedFactors_3 3,3,3,3,3,3,3,3,3,3;
        SpeedFactors_4 3,3,3,3,3,3,3,3,3,3;
        Para4 7,500,630,640,6;

        RETURN;
        MoveL p630, v500, z1, currentTool\WObj:=currentWorkObject;
        MoveL p631, v500, z1, currentTool\WObj:=currentWorkObject;
        MoveL p632, v500, z1, currentTool\WObj:=currentWorkObject;
        MoveL p633, v500, z1, currentTool\WObj:=currentWorkObject;
		MoveL p634, v500, z1, currentTool\WObj:=currentWorkObject;
		MoveL p635, v500, z1, currentTool\WObj:=currentWorkObject;
        !MoveL p636, v500, z1, currentTool\WObj:=currentWorkObject;
		!MoveL p637, v500, z1, currentTool\WObj:=currentWorkObject;
		!MoveL p638, v500, z1, currentTool\WObj:=currentWorkObject;
        !MoveL p639, v500, z1, currentTool\WObj:=currentWorkObject;

        MoveL p640, v500, z1, currentTool\WObj:=currentWorkObject;
        MoveL p641, v500, z1, currentTool\WObj:=currentWorkObject;
        MoveL p642, v500, z1, currentTool\WObj:=currentWorkObject;
        MoveL p643, v500, z1, currentTool\WObj:=currentWorkObject;
		MoveL p644, v500, z1, currentTool\WObj:=currentWorkObject;
		MoveL p645, v500, z1, currentTool\WObj:=currentWorkObject;
		!MoveL p646, v500, z1, currentTool\WObj:=currentWorkObject;
		!MoveL p647, v500, z1, currentTool\WObj:=currentWorkObject;
		!MoveL p648, v500, z1, currentTool\WObj:=currentWorkObject;
        !MoveL p649, v500, z1, currentTool\WObj:=currentWorkObject;


	ENDPROC
    PROC Shroud4()
		MoveL mypounce220, v1000, z50, currentTool\WObj:=currentWorkObject;

        SpeedFactors_3 3,3,3,3,3,3,3,3,3,3;
        SpeedFactors_4 3,3,3,3,3,3,3,3,3,3;
        Para4 7,500,262,268,5;
		MoveL mypounce240, v1000, z50, currentTool\WObj:=currentWorkObject;
		MoveL mypounce250, v1000, z50, currentTool\WObj:=currentWorkObject;

        RETURN;
        MoveL p262, v500, z1, currentTool\WObj:=currentWorkObject;
        MoveL p263, v500, z1, currentTool\WObj:=currentWorkObject;
        MoveL p264, v500, z1, currentTool\WObj:=currentWorkObject;
        MoveL p265, v500, z1, currentTool\WObj:=currentWorkObject;
		MoveL p266, v500, z1, currentTool\WObj:=currentWorkObject;
		!MoveL p267, v500, z1, currentTool\WObj:=currentWorkObject;

        MoveL p268, v500, z1, currentTool\WObj:=currentWorkObject;
		MoveL p269, v500, z1, currentTool\WObj:=currentWorkObject;
		MoveL p270, v500, z1, currentTool\WObj:=currentWorkObject;
        MoveL p271, v500, z1, currentTool\WObj:=currentWorkObject;
		MoveL p272, v500, z1, currentTool\WObj:=currentWorkObject;
		!MoveL p273, v500, z1, currentTool\WObj:=currentWorkObject;


	ENDPROC


ENDMODULE
